LIN {X 0,Y 474.587,Z 340.988,A -85,B 0,C 180,E1 -7401.729,E2 -7401.729} C_VEL
LIN {X 0,Y 474.649,Z 340.986,A -85,B 0,C 180,E1 -7404.494,E2 -7404.494} C_VEL
LIN {X 0,Y 474.672,Z 340.979,A -85,B 0,C 180,E1 -7407.333,E2 -7407.333} C_VEL
LIN {X 0,Y 474.604,Z 340.989,A -85,B 0,C 180,E1 -7410.231,E2 -7410.231} C_VEL
LIN {X 0,Y 474.642,Z 340.983,A -85,B 0,C 180,E1 -7413.221,E2 -7413.221} C_VEL
LIN {X 0,Y 474.592,Z 340.992,A -85,B 0,C 180,E1 -7416.324,E2 -7416.324} C_VEL
LIN {X 0,Y 474.612,Z 340.985,A -85,B 0,C 180,E1 -7419.646,E2 -7419.646} C_VEL
LIN {X 0,Y 474.599,Z 340.99,A -85,B 0,C 180,E1 -7422.234,E2 -7422.234} C_VEL
LIN {X 0,Y 474.616,Z 340.986,A -85,B 0,C 180,E1 -7425.298,E2 -7425.298} C_VEL
LIN {X 0,Y 474.615,Z 340.989,A -85,B 0,C 180,E1 -7428.215,E2 -7428.215} C_VEL
LIN {X 0,Y 474.611,Z 340.986,A -85,B 0,C 180,E1 -7431.543,E2 -7431.543} C_VEL
LIN {X 0,Y 474.623,Z 340.989,A -85,B 0,C 180,E1 -7434.726,E2 -7434.726} C_VEL
LIN {X 0,Y 474.637,Z 340.983,A -85,B 0,C 180,E1 -7437.788,E2 -7437.788} C_VEL
LIN {X 0,Y 474.608,Z 340.989,A -85,B 0,C 180,E1 -7440.889,E2 -7440.889} C_VEL
LIN {X 0,Y 474.612,Z 340.986,A -85,B 0,C 180,E1 -7443.626,E2 -7443.626} C_VEL
LIN {X 0,Y 474.637,Z 340.988,A -85,B 0,C 180,E1 -7446.643,E2 -7446.643} C_VEL
LIN {X 0,Y 474.654,Z 340.984,A -85,B 0,C 180,E1 -7450.09,E2 -7450.09} C_VEL
LIN {X 0,Y 474.642,Z 340.982,A -85,B 0,C 180,E1 -7451.675,E2 -7451.675} C_VEL
LIN {X 0,Y 473.965,Z 341.075,A -85,B 0,C 180,E1 -7452.383,E2 -7452.383} C_VEL
LIN {X 0,Y 471.115,Z 341.424,A -85,B 0,C 180,E1 -7453.534,E2 -7453.534} C_VEL
LIN {X 0,Y 468.709,Z 341.728,A -85,B 0,C 180,E1 -7454.462,E2 -7454.462} C_VEL
LIN {X 0,Y 467.674,Z 341.851,A -85,B 0,C 180,E1 -7455.179,E2 -7455.179} C_VEL
LIN {X 0,Y 467.588,Z 341.86,A -85,B 0,C 180,E1 -7455.422,E2 -7455.422} C_VEL
LIN {X 0,Y 467.653,Z 341.855,A -85,B 0,C 180,E1 -7458.734,E2 -7458.734} C_VEL
LIN {X 0,Y 467.66,Z 341.851,A -85,B 0,C 180,E1 -7461.357,E2 -7461.357} C_VEL
LIN {X 0,Y 467.705,Z 341.85,A -85,B 0,C 180,E1 -7463.963,E2 -7463.963} C_VEL
LIN {X 0,Y 467.817,Z 341.832,A -85,B 0,C 180,E1 -7467.417,E2 -7467.417} C_VEL
LIN {X 0,Y 467.853,Z 341.832,A -85,B 0,C 180,E1 -7470,E2 -7470} C_VEL
LIN {X 0,Y 467.815,Z 341.836,A -85,B 0,C 180,E1 -7472.584,E2 -7472.584} C_VEL
LIN {X 0,Y 467.706,Z 341.852,A -85,B 0,C 180,E1 -7476.038,E2 -7476.038} C_VEL
LIN {X 0,Y 467.637,Z 341.857,A -85,B 0,C 180,E1 -7478.644,E2 -7478.644} C_VEL
LIN {X 0,Y 467.656,Z 341.857,A -85,B 0,C 180,E1 -7482.356,E2 -7482.356} C_VEL
LIN {X 0,Y 467.613,Z 341.978,A -85,B 0,C 180,E1 -7485.194,E2 -7485.194} C_VEL
LIN {X 0,Y 468.283,Z 345.088,A -85,B 0,C 180,E1 -7485.805,E2 -7485.805} C_VEL
LIN {X 0,Y 476.001,Z 364.043,A -85,B 0,C 180,E1 -7486.537,E2 -7486.537} C_VEL
LIN {X 0,Y 474.194,Z 509.031,A -85,B 0,C 180,E1 -7488.849,E2 -7488.849} C_VEL
LIN {X 0,Y 473.785,Z 524.801,A -85,B 0,C 180,E1 -7489.272,E2 -7489.272} C_VEL
LIN {X 0,Y 473.25,Z 539.852,A -85,B 0,C 180,E1 -7489.859,E2 -7489.859} C_VEL
LIN {X 0,Y 472.524,Z 554.963,A -85,B 0,C 180,E1 -7490.645,E2 -7490.645} C_VEL
LIN {X 0,Y 471.782,Z 568.297,A -85,B 0,C 180,E1 -7491.521,E2 -7491.521} C_VEL
LIN {X 0,Y 470.984,Z 580.882,A -85,B 0,C 180,E1 -7492.531,E2 -7492.531} C_VEL
LIN {X 0,Y 470.089,Z 593.972,A -85,B 0,C 180,E1 -7493.808,E2 -7493.808} C_VEL
LIN {X 0,Y 469.383,Z 604.338,A -85,B 0,C 180,E1 -7495.023,E2 -7495.023} C_VEL
LIN {X 0,Y 468.643,Z 615.056,A -85,B 0,C 180,E1 -7496.518,E2 -7496.518} C_VEL
LIN {X 0,Y 468.075,Z 623.773,A -85,B 0,C 180,E1 -7497.983,E2 -7497.983} C_VEL
LIN {X 0,Y 467.53,Z 632.422,A -85,B 0,C 180,E1 -7499.74,E2 -7499.74} C_VEL
LIN {X 0,Y 467.23,Z 638.758,A -85,B 0,C 180,E1 -7501.339,E2 -7501.339} C_VEL
LIN {X 0,Y 466.974,Z 643.497,A -85,B 0,C 180,E1 -7502.807,E2 -7502.807} C_VEL
LIN {X 0,Y 466.851,Z 646.899,A -85,B 0,C 180,E1 -7504.108,E2 -7504.108} C_VEL
LIN {X 0,Y 466.652,Z 650.524,A -85,B 0,C 180,E1 -7505.97,E2 -7505.97} C_VEL
LIN {X 0,Y 466.583,Z 652.01,A -85,B 0,C 180,E1 -7507.05,E2 -7507.05} C_VEL
LIN {X 0,Y 466.575,Z 653.213,A -85,B 0,C 180,E1 -7508.438,E2 -7508.438} C_VEL
LIN {X 0,Y 466.553,Z 653.709,A -85,B 0,C 180,E1 -7510.372,E2 -7510.372} C_VEL
LIN {X 0,Y 466.566,Z 653.334,A -85,B 0,C 180,E1 -7511.513,E2 -7511.513} C_VEL
LIN {X 0,Y 466.619,Z 652.463,A -85,B 0,C 180,E1 -7512.67,E2 -7512.67} C_VEL
LIN {X 0,Y 466.668,Z 651.066,A -85,B 0,C 180,E1 -7513.849,E2 -7513.849} C_VEL
LIN {X 0,Y 466.855,Z 647.895,A -85,B 0,C 180,E1 -7515.607,E2 -7515.607} C_VEL
LIN {X 0,Y 467.042,Z 643.061,A -85,B 0,C 180,E1 -7517.506,E2 -7517.506} C_VEL
LIN {X 0,Y 467.29,Z 637.214,A -85,B 0,C 180,E1 -7519.243,E2 -7519.243} C_VEL
LIN {X 0,Y 467.708,Z 630.356,A -85,B 0,C 180,E1 -7520.867,E2 -7520.867} C_VEL
LIN {X 0,Y 468.244,Z 622.555,A -85,B 0,C 180,E1 -7522.387,E2 -7522.387} C_VEL
LIN {X 0,Y 468.831,Z 613.461,A -85,B 0,C 180,E1 -7523.868,E2 -7523.868} C_VEL
LIN {X 0,Y 469.603,Z 602.591,A -85,B 0,C 180,E1 -7525.34,E2 -7525.34} C_VEL
LIN {X 0,Y 470.454,Z 590.958,A -85,B 0,C 180,E1 -7526.647,E2 -7526.647} C_VEL
LIN {X 0,Y 471.237,Z 578.375,A -85,B 0,C 180,E1 -7527.824,E2 -7527.824} C_VEL
LIN {X 0,Y 472.024,Z 565.723,A -85,B 0,C 180,E1 -7528.798,E2 -7528.798} C_VEL
LIN {X 0,Y 472.796,Z 551.391,A -85,B 0,C 180,E1 -7529.691,E2 -7529.691} C_VEL
LIN {X 0,Y 473.431,Z 537.673,A -85,B 0,C 180,E1 -7530.362,E2 -7530.362} C_VEL
LIN {X 0,Y 473.882,Z 522.925,A -85,B 0,C 180,E1 -7530.909,E2 -7530.909} C_VEL
LIN {X 0,Y 474.283,Z 507.871,A -85,B 0,C 180,E1 -7531.288,E2 -7531.288} C_VEL
LIN {X 0,Y 476.111,Z 364.185,A -85,B 0,C 180,E1 -7533.601,E2 -7533.601} C_VEL
LIN {X 0,Y 468.631,Z 346.42,A -85,B 0,C 180,E1 -7534.341,E2 -7534.341} C_VEL
LIN {X 0,Y 467.593,Z 341.868,A -85,B 0,C 180,E1 -7535.29,E2 -7535.29} C_VEL
LIN {X 0,Y 467.573,Z 341.864,A -85,B 0,C 180,E1 -7538.854,E2 -7538.854} C_VEL
LIN {X 0,Y 467.621,Z 341.863,A -85,B 0,C 180,E1 -7541.602,E2 -7541.602} C_VEL
LIN {X 0,Y 467.598,Z 341.864,A -85,B 0,C 180,E1 -7545.196,E2 -7545.196} C_VEL
LIN {X 0,Y 467.66,Z 341.859,A -85,B 0,C 180,E1 -7547.854,E2 -7547.854} C_VEL
LIN {X 0,Y 467.66,Z 341.857,A -85,B 0,C 180,E1 -7551.356,E2 -7551.356} C_VEL
LIN {X 0,Y 467.706,Z 341.851,A -85,B 0,C 180,E1 -7553.962,E2 -7553.962} C_VEL
LIN {X 0,Y 467.817,Z 341.837,A -85,B 0,C 180,E1 -7557.417,E2 -7557.417} C_VEL
LIN {X 0,Y 467.881,Z 341.829,A -85,B 0,C 180,E1 -7560,E2 -7560} C_VEL
LIN {X 0,Y 467.853,Z 341.828,A -85,B 0,C 180,E1 -7562.583,E2 -7562.583} C_VEL
LIN {X 0,Y 467.715,Z 341.847,A -85,B 0,C 180,E1 -7566.037,E2 -7566.037} C_VEL
LIN {X 0,Y 467.67,Z 341.852,A -85,B 0,C 180,E1 -7568.643,E2 -7568.643} C_VEL
LIN {X 0,Y 467.659,Z 341.852,A -85,B 0,C 180,E1 -7572.145,E2 -7572.145} C_VEL
LIN {X 0,Y 467.641,Z 341.856,A -85,B 0,C 180,E1 -7575.695,E2 -7575.695} C_VEL
LIN {X 0,Y 467.624,Z 341.861,A -85,B 0,C 180,E1 -7579.307,E2 -7579.307} C_VEL
LIN {X 0,Y 467.536,Z 341.868,A -85,B 0,C 180,E1 -7582.073,E2 -7582.073} C_VEL
LIN {X 0,Y 467.603,Z 341.861,A -85,B 0,C 180,E1 -7584.887,E2 -7584.887} C_VEL
LIN {X 0,Y 467.622,Z 341.859,A -85,B 0,C 180,E1 -7587.769,E2 -7587.769} C_VEL
LIN {X 0,Y 467.57,Z 341.87,A -85,B 0,C 180,E1 -7591.045,E2 -7591.045} C_VEL
LIN {X 0,Y 467.589,Z 341.863,A -85,B 0,C 180,E1 -7594.242,E2 -7594.242} C_VEL
LIN {X 0,Y 467.549,Z 341.872,A -85,B 0,C 180,E1 -7597.186,E2 -7597.186} C_VEL
LIN {X 0,Y 467.579,Z 341.865,A -85,B 0,C 180,E1 -7600.264,E2 -7600.264} C_VEL
LIN {X 0,Y 467.588,Z 341.867,A -85,B 0,C 180,E1 -7602.567,E2 -7602.567} C_VEL
LIN {X 0,Y 467.572,Z 341.87,A -85,B 0,C 180,E1 -7605.053,E2 -7605.053} C_VEL
LIN {X 0,Y 467.59,Z 341.865,A -85,B 0,C 180,E1 -7607.44,E2 -7607.44} C_VEL
LIN {X 0,Y 467.583,Z 341.866,A -85,B 0,C 180,E1 -7610.855,E2 -7610.855} C_VEL
LIN {X 0,Y 467.561,Z 341.87,A -85,B 0,C 180,E1 -7614.261,E2 -7614.261} C_VEL
LIN {X 0,Y 467.583,Z 341.869,A -85,B 0,C 180,E1 -7617.321,E2 -7617.321} C_VEL
LIN {X 0,Y 467.59,Z 341.957,A -85,B 0,C 180,E1 -7618.29,E2 -7618.29} C_VEL
LIN {X 0,Y 470.988,Z 355.341,A -85,B 0,C 180,E1 -7620.5,E2 -7620.5} C_VEL
LIN {X 0,Y 472.508,Z 362.159,A -85,B 0,C 180,E1 -7621.578,E2 -7621.578} C_VEL
LIN {X 0,Y 472.251,Z 370.532,A -85,B 0,C 180,E1 -7622.758,E2 -7622.758} C_VEL
LIN {X 0,Y 471.054,Z 392.478,A -85,B 0,C 180,E1 -7625.776,E2 -7625.776} C_VEL
LIN {X 0,Y 471.112,Z 393.337,A -85,B 0,C 180,E1 -7625.837,E2 -7625.837} C_VEL
LIN {X 0,Y 475.725,Z 419.308,A -85,B 0,C 180,E1 -7626.526,E2 -7626.526} C_VEL
LIN {X 0,Y 473.906,Z 560.263,A -85,B 0,C 180,E1 -7628.78,E2 -7628.78} C_VEL
LIN {X 0,Y 473.379,Z 576.364,A -85,B 0,C 180,E1 -7629.212,E2 -7629.212} C_VEL
LIN {X 0,Y 472.664,Z 591.498,A -85,B 0,C 180,E1 -7629.797,E2 -7629.797} C_VEL
LIN {X 0,Y 471.905,Z 605.905,A -85,B 0,C 180,E1 -7630.535,E2 -7630.535} C_VEL
LIN {X 0,Y 471.102,Z 619.398,A -85,B 0,C 180,E1 -7631.405,E2 -7631.405} C_VEL
LIN {X 0,Y 470.194,Z 633.159,A -85,B 0,C 180,E1 -7632.493,E2 -7632.493} C_VEL
LIN {X 0,Y 469.381,Z 645.67,A -85,B 0,C 180,E1 -7633.695,E2 -7633.695} C_VEL
LIN {X 0,Y 468.624,Z 657.082,A -85,B 0,C 180,E1 -7635.007,E2 -7635.007} C_VEL
LIN {X 0,Y 468.004,Z 668.188,A -85,B 0,C 180,E1 -7636.54,E2 -7636.54} C_VEL
LIN {X 0,Y 467.478,Z 677.417,A -85,B 0,C 180,E1 -7638.07,E2 -7638.07} C_VEL
LIN {X 0,Y 467.199,Z 685.087,A -85,B 0,C 180,E1 -7639.6,E2 -7639.6} C_VEL
LIN {X 0,Y 466.898,Z 692.25,A -85,B 0,C 180,E1 -7641.342,E2 -7641.342} C_VEL
LIN {X 0,Y 466.818,Z 697.893,A -85,B 0,C 180,E1 -7643.082,E2 -7643.082} C_VEL
LIN {X 0,Y 466.711,Z 702.161,A -85,B 0,C 180,E1 -7644.816,E2 -7644.816} C_VEL
LIN {X 0,Y 466.708,Z 705.163,A -85,B 0,C 180,E1 -7646.546,E2 -7646.546} C_VEL
LIN {X 0,Y 466.692,Z 706.959,A -85,B 0,C 180,E1 -7648.274,E2 -7648.274} C_VEL
LIN {X 0,Y 466.596,Z 707.583,A -85,B 0,C 180,E1 -7650,E2 -7650} C_VEL
LIN {X 0,Y 466.691,Z 706.998,A -85,B 0,C 180,E1 -7651.726,E2 -7651.726} C_VEL
LIN {X 0,Y 466.707,Z 705.239,A -85,B 0,C 180,E1 -7653.453,E2 -7653.453} C_VEL
LIN {X 0,Y 466.708,Z 702.281,A -85,B 0,C 180,E1 -7655.183,E2 -7655.183} C_VEL
LIN {X 0,Y 466.729,Z 698.058,A -85,B 0,C 180,E1 -7656.918,E2 -7656.918} C_VEL
LIN {X 0,Y 466.898,Z 692.464,A -85,B 0,C 180,E1 -7658.657,E2 -7658.657} C_VEL
LIN {X 0,Y 467.201,Z 685.346,A -85,B 0,C 180,E1 -7660.399,E2 -7660.399} C_VEL
LIN {X 0,Y 467.515,Z 677.733,A -85,B 0,C 180,E1 -7661.929,E2 -7661.929} C_VEL
LIN {X 0,Y 468.043,Z 668.563,A -85,B 0,C 180,E1 -7663.458,E2 -7663.458} C_VEL
LIN {X 0,Y 468.655,Z 657.51,A -85,B 0,C 180,E1 -7664.991,E2 -7664.991} C_VEL
LIN {X 0,Y 469.442,Z 646.16,A -85,B 0,C 180,E1 -7666.302,E2 -7666.302} C_VEL
LIN {X 0,Y 470.221,Z 633.697,A -85,B 0,C 180,E1 -7667.505,E2 -7667.505} C_VEL
LIN {X 0,Y 471.129,Z 619.955,A -85,B 0,C 180,E1 -7668.593,E2 -7668.593} C_VEL
LIN {X 0,Y 471.948,Z 606.475,A -85,B 0,C 180,E1 -7669.462,E2 -7669.462} C_VEL
LIN {X 0,Y 472.758,Z 592.065,A -85,B 0,C 180,E1 -7670.199,E2 -7670.199} C_VEL
LIN {X 0,Y 473.357,Z 576.997,A -85,B 0,C 180,E1 -7670.785,E2 -7670.785} C_VEL
LIN {X 0,Y 473.904,Z 561.89,A -85,B 0,C 180,E1 -7671.191,E2 -7671.191} C_VEL
LIN {X 0,Y 475.392,Z 446.29,A -85,B 0,C 180,E1 -7673.034,E2 -7673.034} C_VEL
LIN {X 0,Y 475.685,Z 419.152,A -85,B 0,C 180,E1 -7673.468,E2 -7673.468} C_VEL
LIN {X 0,Y 471.151,Z 394.04,A -85,B 0,C 180,E1 -7674.124,E2 -7674.124} C_VEL
LIN {X 0,Y 472.402,Z 371.288,A -85,B 0,C 180,E1 -7677.241,E2 -7677.241} C_VEL
LIN {X 0,Y 472.755,Z 362.946,A -85,B 0,C 180,E1 -7678.405,E2 -7678.405} C_VEL
LIN {X 0,Y 468.809,Z 346.686,A -85,B 0,C 180,E1 -7680.998,E2 -7680.998} C_VEL
LIN {X 0,Y 467.572,Z 341.869,A -85,B 0,C 180,E1 -7681.804,E2 -7681.804} C_VEL
LIN {X 0,Y 467.562,Z 341.87,A -85,B 0,C 180,E1 -7684.832,E2 -7684.832} C_VEL
LIN {X 0,Y 467.563,Z 341.87,A -85,B 0,C 180,E1 -7688.044,E2 -7688.044} C_VEL
LIN {X 0,Y 467.579,Z 341.87,A -85,B 0,C 180,E1 -7691.277,E2 -7691.277} C_VEL
LIN {X 0,Y 467.564,Z 341.865,A -85,B 0,C 180,E1 -7693.822,E2 -7693.822} C_VEL
LIN {X 0,Y 467.568,Z 341.863,A -85,B 0,C 180,E1 -7696.257,E2 -7696.257} C_VEL
LIN {X 0,Y 467.579,Z 341.864,A -85,B 0,C 180,E1 -7698.722,E2 -7698.722} C_VEL
LIN {X 0,Y 467.563,Z 341.864,A -85,B 0,C 180,E1 -7701.956,E2 -7701.956} C_VEL
LIN {X 0,Y 467.566,Z 341.872,A -85,B 0,C 180,E1 -7705.168,E2 -7705.168} C_VEL
LIN {X 0,Y 467.579,Z 341.862,A -85,B 0,C 180,E1 -7708.26,E2 -7708.26} C_VEL
LIN {X 0,Y 467.574,Z 341.869,A -85,B 0,C 180,E1 -7711.251,E2 -7711.251} C_VEL
LIN {X 0,Y 467.607,Z 341.858,A -85,B 0,C 180,E1 -7714.16,E2 -7714.16} C_VEL
LIN {X 0,Y 467.574,Z 341.87,A -85,B 0,C 180,E1 -7716.996,E2 -7716.996} C_VEL
LIN {X 0,Y 467.621,Z 341.857,A -85,B 0,C 180,E1 -7719.777,E2 -7719.777} C_VEL
LIN {X 0,Y 467.606,Z 341.86,A -85,B 0,C 180,E1 -7722.507,E2 -7722.507} C_VEL
LIN {X 0,Y 467.605,Z 341.864,A -85,B 0,C 180,E1 -7725.197,E2 -7725.197} C_VEL
LIN {X 0,Y 467.653,Z 341.852,A -85,B 0,C 180,E1 -7727.855,E2 -7727.855} C_VEL
LIN {X 0,Y 467.679,Z 341.852,A -85,B 0,C 180,E1 -7731.357,E2 -7731.357} C_VEL
LIN {X 0,Y 467.732,Z 341.842,A -85,B 0,C 180,E1 -7733.963,E2 -7733.963} C_VEL
LIN {X 0,Y 467.858,Z 341.829,A -85,B 0,C 180,E1 -7737.417,E2 -7737.417} C_VEL
LIN {X 0,Y 467.881,Z 341.824,A -85,B 0,C 180,E1 -7740,E2 -7740} C_VEL
LIN {X 0,Y 467.857,Z 341.831,A -85,B 0,C 180,E1 -7742.583,E2 -7742.583} C_VEL
LIN {X 0,Y 467.744,Z 341.841,A -85,B 0,C 180,E1 -7746.038,E2 -7746.038} C_VEL
LIN {X 0,Y 467.68,Z 341.855,A -85,B 0,C 180,E1 -7748.643,E2 -7748.643} C_VEL
LIN {X 0,Y 467.654,Z 341.853,A -85,B 0,C 180,E1 -7752.146,E2 -7752.146} C_VEL
LIN {X 0,Y 467.637,Z 341.854,A -85,B 0,C 180,E1 -7755.695,E2 -7755.695} C_VEL
LIN {X 0,Y 467.616,Z 341.866,A -85,B 0,C 180,E1 -7758.765,E2 -7758.765} C_VEL
LIN {X 0,Y 467.579,Z 341.864,A -85,B 0,C 180,E1 -7761.269,E2 -7761.269} C_VEL
LIN {X 0,Y 467.567,Z 341.863,A -85,B 0,C 180,E1 -7763.944,E2 -7763.944} C_VEL
LIN {X 0,Y 467.589,Z 341.868,A -85,B 0,C 180,E1 -7766.802,E2 -7766.802} C_VEL
LIN {X 0,Y 467.552,Z 341.865,A -85,B 0,C 180,E1 -7769.739,E2 -7769.739} C_VEL
LIN {X 0,Y 467.582,Z 341.868,A -85,B 0,C 180,E1 -7772.759,E2 -7772.759} C_VEL
LIN {X 0,Y 467.555,Z 341.865,A -85,B 0,C 180,E1 -7775.89,E2 -7775.89} C_VEL
LIN {X 0,Y 467.557,Z 341.866,A -85,B 0,C 180,E1 -7779.148,E2 -7779.148} C_VEL
LIN {X 0,Y 467.572,Z 341.863,A -85,B 0,C 180,E1 -7781.404,E2 -7781.404} C_VEL
LIN {X 0,Y 467.565,Z 341.866,A -85,B 0,C 180,E1 -7785.053,E2 -7785.053} C_VEL
LIN {X 0,Y 467.574,Z 341.87,A -85,B 0,C 180,E1 -7788.597,E2 -7788.597} C_VEL
LIN {X 0,Y 467.563,Z 341.865,A -85,B 0,C 180,E1 -7791.956,E2 -7791.956} C_VEL
LIN {X 0,Y 467.564,Z 341.864,A -85,B 0,C 180,E1 -7795.168,E2 -7795.168} C_VEL
LIN {X 0,Y 467.584,Z 341.866,A -85,B 0,C 180,E1 -7798.261,E2 -7798.261} C_VEL
LIN {X 0,Y 467.557,Z 341.865,A -85,B 0,C 180,E1 -7801.25,E2 -7801.25} C_VEL
LIN {X 0,Y 467.584,Z 341.865,A -85,B 0,C 180,E1 -7804.159,E2 -7804.159} C_VEL
LIN {X 0,Y 467.578,Z 341.863,A -85,B 0,C 180,E1 -7806.996,E2 -7806.996} C_VEL
LIN {X 0,Y 467.623,Z 341.857,A -85,B 0,C 180,E1 -7809.778,E2 -7809.778} C_VEL
LIN {X 0,Y 467.571,Z 341.869,A -85,B 0,C 180,E1 -7812.506,E2 -7812.506} C_VEL
LIN {X 0,Y 467.588,Z 341.86,A -85,B 0,C 180,E1 -7815.422,E2 -7815.422} C_VEL
LIN {X 0,Y 466.921,Z 341.95,A -85,B 0,C 180,E1 -7816.141,E2 -7816.141} C_VEL
LIN {X 0,Y 464.082,Z 342.299,A -85,B 0,C 180,E1 -7817.31,E2 -7817.31} C_VEL
LIN {X 0,Y 461.684,Z 342.603,A -85,B 0,C 180,E1 -7818.252,E2 -7818.252} C_VEL
LIN {X 0,Y 460.657,Z 342.725,A -85,B 0,C 180,E1 -7818.98,E2 -7818.98} C_VEL
LIN {X 0,Y 460.574,Z 342.734,A -85,B 0,C 180,E1 -7819.226,E2 -7819.226} C_VEL
LIN {X 0,Y 460.667,Z 342.727,A -85,B 0,C 180,E1 -7822.594,E2 -7822.594} C_VEL
LIN {X 0,Y 460.677,Z 342.724,A -85,B 0,C 180,E1 -7824.748,E2 -7824.748} C_VEL
LIN {X 0,Y 460.761,Z 342.711,A -85,B 0,C 180,E1 -7827.378,E2 -7827.378} C_VEL
LIN {X 0,Y 460.823,Z 342.708,A -85,B 0,C 180,E1 -7830,E2 -7830} C_VEL
LIN {X 0,Y 460.759,Z 342.714,A -85,B 0,C 180,E1 -7832.623,E2 -7832.623} C_VEL
LIN {X 0,Y 460.672,Z 342.729,A -85,B 0,C 180,E1 -7836.131,E2 -7836.131} C_VEL
LIN {X 0,Y 460.592,Z 342.733,A -85,B 0,C 180,E1 -7838.777,E2 -7838.777} C_VEL
LIN {X 0,Y 460.602,Z 342.735,A -85,B 0,C 180,E1 -7842.435,E2 -7842.435} C_VEL
LIN {X 0,Y 460.552,Z 342.857,A -85,B 0,C 180,E1 -7844.895,E2 -7844.895} C_VEL
LIN {X 0,Y 461.146,Z 345.416,A -85,B 0,C 180,E1 -7845.412,E2 -7845.412} C_VEL
LIN {X 0,Y 469.499,Z 365.897,A -85,B 0,C 180,E1 -7846.226,E2 -7846.226} C_VEL
LIN {X 0,Y 467.558,Z 509.675,A -85,B 0,C 180,E1 -7848.554,E2 -7848.554} C_VEL
LIN {X 0,Y 467.13,Z 525.283,A -85,B 0,C 180,E1 -7848.981,E2 -7848.981} C_VEL
LIN {X 0,Y 466.554,Z 540.472,A -85,B 0,C 180,E1 -7849.583,E2 -7849.583} C_VEL
LIN {X 0,Y 465.902,Z 554.198,A -85,B 0,C 180,E1 -7850.301,E2 -7850.301} C_VEL
LIN {X 0,Y 465.084,Z 567.53,A -85,B 0,C 180,E1 -7851.173,E2 -7851.173} C_VEL
LIN {X 0,Y 464.192,Z 580.845,A -85,B 0,C 180,E1 -7852.242,E2 -7852.242} C_VEL
LIN {X 0,Y 463.362,Z 593.316,A -85,B 0,C 180,E1 -7853.463,E2 -7853.463} C_VEL
LIN {X 0,Y 462.556,Z 603.963,A -85,B 0,C 180,E1 -7854.71,E2 -7854.71} C_VEL
LIN {X 0,Y 461.765,Z 614.583,A -85,B 0,C 180,E1 -7856.192,E2 -7856.192} C_VEL
LIN {X 0,Y 461.203,Z 622.632,A -85,B 0,C 180,E1 -7857.53,E2 -7857.53} C_VEL
LIN {X 0,Y 460.63,Z 631.16,A -85,B 0,C 180,E1 -7859.225,E2 -7859.225} C_VEL
LIN {X 0,Y 460.254,Z 637.429,A -85,B 0,C 180,E1 -7860.735,E2 -7860.735} C_VEL
LIN {X 0,Y 459.985,Z 642.836,A -85,B 0,C 180,E1 -7862.328,E2 -7862.328} C_VEL
LIN {X 0,Y 459.79,Z 646.935,A -85,B 0,C 180,E1 -7863.87,E2 -7863.87} C_VEL
LIN {X 0,Y 459.619,Z 650.289,A -85,B 0,C 180,E1 -7865.525,E2 -7865.525} C_VEL
LIN {X 0,Y 459.48,Z 652.728,A -85,B 0,C 180,E1 -7867.309,E2 -7867.309} C_VEL
LIN {X 0,Y 459.472,Z 653.857,A -85,B 0,C 180,E1 -7868.839,E2 -7868.839} C_VEL
LIN {X 0,Y 459.463,Z 654.164,A -85,B 0,C 180,E1 -7870.11,E2 -7870.11} C_VEL
LIN {X 0,Y 459.478,Z 653.79,A -85,B 0,C 180,E1 -7871.454,E2 -7871.454} C_VEL
LIN {X 0,Y 459.545,Z 652.825,A -85,B 0,C 180,E1 -7872.77,E2 -7872.77} C_VEL
LIN {X 0,Y 459.695,Z 650.23,A -85,B 0,C 180,E1 -7874.69,E2 -7874.69} C_VEL
LIN {X 0,Y 459.889,Z 646.337,A -85,B 0,C 180,E1 -7876.552,E2 -7876.552} C_VEL
LIN {X 0,Y 460.131,Z 640.885,A -85,B 0,C 180,E1 -7878.454,E2 -7878.454} C_VEL
LIN {X 0,Y 460.476,Z 634.689,A -85,B 0,C 180,E1 -7880.131,E2 -7880.131} C_VEL
LIN {X 0,Y 460.892,Z 628.162,A -85,B 0,C 180,E1 -7881.582,E2 -7881.582} C_VEL
LIN {X 0,Y 461.469,Z 620.506,A -85,B 0,C 180,E1 -7883.017,E2 -7883.017} C_VEL
LIN {X 0,Y 462.129,Z 611.26,A -85,B 0,C 180,E1 -7884.473,E2 -7884.473} C_VEL
LIN {X 0,Y 462.951,Z 600.977,A -85,B 0,C 180,E1 -7885.827,E2 -7885.827} C_VEL
LIN {X 0,Y 463.773,Z 589.761,A -85,B 0,C 180,E1 -7887.067,E2 -7887.067} C_VEL
LIN {X 0,Y 464.547,Z 578.052,A -85,B 0,C 180,E1 -7888.155,E2 -7888.155} C_VEL
LIN {X 0,Y 465.38,Z 565.74,A -85,B 0,C 180,E1 -7889.105,E2 -7889.105} C_VEL
LIN {X 0,Y 466.139,Z 551.782,A -85,B 0,C 180,E1 -7889.984,E2 -7889.984} C_VEL
LIN {X 0,Y 466.842,Z 537.238,A -85,B 0,C 180,E1 -7890.699,E2 -7890.699} C_VEL
LIN {X 0,Y 467.344,Z 521.749,A -85,B 0,C 180,E1 -7891.265,E2 -7891.265} C_VEL
LIN {X 0,Y 467.724,Z 506.873,A -85,B 0,C 180,E1 -7891.627,E2 -7891.627} C_VEL
LIN {X 0,Y 469.739,Z 366.212,A -85,B 0,C 180,E1 -7893.922,E2 -7893.922} C_VEL
LIN {X 0,Y 462.361,Z 349.033,A -85,B 0,C 180,E1 -7894.656,E2 -7894.656} C_VEL
LIN {X 0,Y 461.525,Z 346.887,A -85,B 0,C 180,E1 -7894.762,E2 -7894.762} C_VEL
LIN {X 0,Y 460.541,Z 342.744,A -85,B 0,C 180,E1 -7895.667,E2 -7895.667} C_VEL
LIN {X 0,Y 460.52,Z 342.743,A -85,B 0,C 180,E1 -7898.58,E2 -7898.58} C_VEL
LIN {X 0,Y 460.585,Z 342.736,A -85,B 0,C 180,E1 -7901.31,E2 -7901.31} C_VEL
LIN {X 0,Y 460.57,Z 342.742,A -85,B 0,C 180,E1 -7904.057,E2 -7904.057} C_VEL
LIN {X 0,Y 460.613,Z 342.736,A -85,B 0,C 180,E1 -7907.666,E2 -7907.666} C_VEL
LIN {X 0,Y 460.612,Z 342.734,A -85,B 0,C 180,E1 -7911.223,E2 -7911.223} C_VEL
LIN {X 0,Y 460.672,Z 342.729,A -85,B 0,C 180,E1 -7913.869,E2 -7913.869} C_VEL
LIN {X 0,Y 460.761,Z 342.716,A -85,B 0,C 180,E1 -7917.377,E2 -7917.377} C_VEL
LIN {X 0,Y 460.851,Z 342.704,A -85,B 0,C 180,E1 -7920,E2 -7920} C_VEL
LIN {X 0,Y 460.794,Z 342.708,A -85,B 0,C 180,E1 -7922.622,E2 -7922.622} C_VEL
LIN {X 0,Y 460.68,Z 342.723,A -85,B 0,C 180,E1 -7926.13,E2 -7926.13} C_VEL
LIN {X 0,Y 460.62,Z 342.731,A -85,B 0,C 180,E1 -7928.776,E2 -7928.776} C_VEL
LIN {X 0,Y 460.616,Z 342.729,A -85,B 0,C 180,E1 -7932.445,E2 -7932.445} C_VEL
LIN {X 0,Y 460.603,Z 342.731,A -85,B 0,C 180,E1 -7935.997,E2 -7935.997} C_VEL
LIN {X 0,Y 460.57,Z 342.74,A -85,B 0,C 180,E1 -7939.615,E2 -7939.615} C_VEL
LIN {X 0,Y 460.512,Z 342.743,A -85,B 0,C 180,E1 -7942.428,E2 -7942.428} C_VEL
LIN {X 0,Y 460.57,Z 342.738,A -85,B 0,C 180,E1 -7945.802,E2 -7945.802} C_VEL
LIN {X 0,Y 460.554,Z 342.738,A -85,B 0,C 180,E1 -7948.233,E2 -7948.233} C_VEL
LIN {X 0,Y 460.523,Z 342.747,A -85,B 0,C 180,E1 -7951.283,E2 -7951.283} C_VEL
LIN {X 0,Y 460.533,Z 342.743,A -85,B 0,C 180,E1 -7954.505,E2 -7954.505} C_VEL
LIN {X 0,Y 460.502,Z 342.748,A -85,B 0,C 180,E1 -7957.623,E2 -7957.623} C_VEL
LIN {X 0,Y 460.543,Z 342.742,A -85,B 0,C 180,E1 -7960.269,E2 -7960.269} C_VEL
LIN {X 0,Y 460.502,Z 342.749,A -85,B 0,C 180,E1 -7963.375,E2 -7963.375} C_VEL
LIN {X 0,Y 460.51,Z 342.748,A -85,B 0,C 180,E1 -7966.625,E2 -7966.625} C_VEL
LIN {X 0,Y 460.544,Z 342.743,A -85,B 0,C 180,E1 -7969.73,E2 -7969.73} C_VEL
LIN {X 0,Y 460.527,Z 342.749,A -85,B 0,C 180,E1 -7972.519,E2 -7972.519} C_VEL
LIN {X 0,Y 460.547,Z 342.743,A -85,B 0,C 180,E1 -7975.623,E2 -7975.623} C_VEL
LIN {X 0,Y 460.573,Z 342.841,A -85,B 0,C 180,E1 -7977.927,E2 -7977.927} C_VEL
LIN {X 0,Y 464.108,Z 356.713,A -85,B 0,C 180,E1 -7980.268,E2 -7980.268} C_VEL
LIN {X 0,Y 465.66,Z 363.48,A -85,B 0,C 180,E1 -7981.363,E2 -7981.363} C_VEL
LIN {X 0,Y 465.683,Z 368.551,A -85,B 0,C 180,E1 -7982.105,E2 -7982.105} C_VEL
LIN {X 0,Y 464.362,Z 390.424,A -85,B 0,C 180,E1 -7985.166,E2 -7985.166} C_VEL
LIN {X 0,Y 464.282,Z 392.309,A -85,B 0,C 180,E1 -7985.429,E2 -7985.429} C_VEL
LIN {X 0,Y 469.206,Z 420.118,A -85,B 0,C 180,E1 -7986.191,E2 -7986.191} C_VEL
LIN {X 0,Y 467.501,Z 547.155,A -85,B 0,C 180,E1 -7988.243,E2 -7988.243} C_VEL
LIN {X 0,Y 467.162,Z 564.361,A -85,B 0,C 180,E1 -7988.574,E2 -7988.574} C_VEL
LIN {X 0,Y 466.567,Z 579.856,A -85,B 0,C 180,E1 -7989.044,E2 -7989.044} C_VEL
LIN {X 0,Y 465.835,Z 593.897,A -85,B 0,C 180,E1 -7989.634,E2 -7989.634} C_VEL
LIN {X 0,Y 464.933,Z 609.002,A -85,B 0,C 180,E1 -7990.461,E2 -7990.461} C_VEL
LIN {X 0,Y 463.969,Z 623.292,A -85,B 0,C 180,E1 -7991.452,E2 -7991.452} C_VEL
LIN {X 0,Y 463.078,Z 636.278,A -85,B 0,C 180,E1 -7992.558,E2 -7992.558} C_VEL
LIN {X 0,Y 462.358,Z 647.201,A -85,B 0,C 180,E1 -7993.667,E2 -7993.667} C_VEL
LIN {X 0,Y 461.54,Z 658.296,A -85,B 0,C 180,E1 -7994.997,E2 -7994.997} C_VEL
LIN {X 0,Y 460.929,Z 669.114,A -85,B 0,C 180,E1 -7996.554,E2 -7996.554} C_VEL
LIN {X 0,Y 460.406,Z 678.194,A -85,B 0,C 180,E1 -7998.121,E2 -7998.121} C_VEL
LIN {X 0,Y 460.127,Z 684.64,A -85,B 0,C 180,E1 -7999.438,E2 -7999.438} C_VEL
LIN {X 0,Y 459.834,Z 691.812,A -85,B 0,C 180,E1 -8001.208,E2 -8001.208} C_VEL
LIN {X 0,Y 459.727,Z 697.463,A -85,B 0,C 180,E1 -8002.975,E2 -8002.975} C_VEL
LIN {X 0,Y 459.619,Z 701.738,A -85,B 0,C 180,E1 -8004.736,E2 -8004.736} C_VEL
LIN {X 0,Y 459.62,Z 704.746,A -85,B 0,C 180,E1 -8006.493,E2 -8006.493} C_VEL
LIN {X 0,Y 459.629,Z 706.549,A -85,B 0,C 180,E1 -8008.247,E2 -8008.247} C_VEL
LIN {X 0,Y 459.527,Z 707.175,A -85,B 0,C 180,E1 -8010,E2 -8010} C_VEL
LIN {X 0,Y 459.628,Z 706.592,A -85,B 0,C 180,E1 -8011.752,E2 -8011.752} C_VEL
LIN {X 0,Y 459.619,Z 704.83,A -85,B 0,C 180,E1 -8013.506,E2 -8013.506} C_VEL
LIN {X 0,Y 459.615,Z 701.87,A -85,B 0,C 180,E1 -8015.264,E2 -8015.264} C_VEL
LIN {X 0,Y 459.652,Z 697.643,A -85,B 0,C 180,E1 -8017.026,E2 -8017.026} C_VEL
LIN {X 0,Y 459.833,Z 692.043,A -85,B 0,C 180,E1 -8018.791,E2 -8018.791} C_VEL
LIN {X 0,Y 460.13,Z 684.917,A -85,B 0,C 180,E1 -8020.561,E2 -8020.561} C_VEL
LIN {X 0,Y 460.482,Z 677.294,A -85,B 0,C 180,E1 -8022.113,E2 -8022.113} C_VEL
LIN {X 0,Y 461.051,Z 668.111,A -85,B 0,C 180,E1 -8023.666,E2 -8023.666} C_VEL
LIN {X 0,Y 461.712,Z 657.035,A -85,B 0,C 180,E1 -8025.222,E2 -8025.222} C_VEL
LIN {X 0,Y 462.539,Z 645.665,A -85,B 0,C 180,E1 -8026.552,E2 -8026.552} C_VEL
LIN {X 0,Y 463.308,Z 633.177,A -85,B 0,C 180,E1 -8027.775,E2 -8027.775} C_VEL
LIN {X 0,Y 464.359,Z 619.409,A -85,B 0,C 180,E1 -8028.875,E2 -8028.875} C_VEL
LIN {X 0,Y 465.189,Z 605.901,A -85,B 0,C 180,E1 -8029.757,E2 -8029.757} C_VEL
LIN {X 0,Y 466.03,Z 591.884,A -85,B 0,C 180,E1 -8030.482,E2 -8030.482} C_VEL
LIN {X 0,Y 466.714,Z 576.352,A -85,B 0,C 180,E1 -8031.093,E2 -8031.093} C_VEL
LIN {X 0,Y 467.254,Z 561.022,A -85,B 0,C 180,E1 -8031.507,E2 -8031.507} C_VEL
LIN {X 0,Y 469.028,Z 431.404,A -85,B 0,C 180,E1 -8033.601,E2 -8033.601} C_VEL
LIN {X 0,Y 469.031,Z 419.626,A -85,B 0,C 180,E1 -8033.8,E2 -8033.8} C_VEL
LIN {X 0,Y 464.389,Z 393.575,A -85,B 0,C 180,E1 -8034.504,E2 -8034.504} C_VEL
LIN {X 0,Y 465.595,Z 372.672,A -85,B 0,C 180,E1 -8037.411,E2 -8037.411} C_VEL
LIN {X 0,Y 465.989,Z 364.902,A -85,B 0,C 180,E1 -8038.51,E2 -8038.51} C_VEL
LIN {X 0,Y 461.89,Z 347.962,A -85,B 0,C 180,E1 -8041.254,E2 -8041.254} C_VEL
LIN {X 0,Y 460.544,Z 342.742,A -85,B 0,C 180,E1 -8042.166,E2 -8042.166} C_VEL
LIN {X 0,Y 460.508,Z 342.748,A -85,B 0,C 180,E1 -8045.445,E2 -8045.445} C_VEL
LIN {X 0,Y 460.542,Z 342.748,A -85,B 0,C 180,E1 -8048.898,E2 -8048.898} C_VEL
LIN {X 0,Y 460.521,Z 342.741,A -85,B 0,C 180,E1 -8052.181,E2 -8052.181} C_VEL
LIN {X 0,Y 460.518,Z 342.747,A -85,B 0,C 180,E1 -8055.412,E2 -8055.412} C_VEL
LIN {X 0,Y 460.532,Z 342.74,A -85,B 0,C 180,E1 -8058.397,E2 -8058.397} C_VEL
LIN {X 0,Y 460.523,Z 342.748,A -85,B 0,C 180,E1 -8061.267,E2 -8061.267} C_VEL
LIN {X 0,Y 460.511,Z 342.743,A -85,B 0,C 180,E1 -8064.555,E2 -8064.555} C_VEL
LIN {X 0,Y 460.528,Z 342.741,A -85,B 0,C 180,E1 -8067.716,E2 -8067.716} C_VEL
LIN {X 0,Y 460.537,Z 342.742,A -85,B 0,C 180,E1 -8070.769,E2 -8070.769} C_VEL
LIN {X 0,Y 460.56,Z 342.737,A -85,B 0,C 180,E1 -8073.735,E2 -8073.735} C_VEL
LIN {X 0,Y 460.543,Z 342.741,A -85,B 0,C 180,E1 -8076.624,E2 -8076.624} C_VEL
LIN {X 0,Y 460.549,Z 342.74,A -85,B 0,C 180,E1 -8079.453,E2 -8079.453} C_VEL
LIN {X 0,Y 460.556,Z 342.737,A -85,B 0,C 180,E1 -8082.23,E2 -8082.23} C_VEL
LIN {X 0,Y 460.563,Z 342.743,A -85,B 0,C 180,E1 -8084.965,E2 -8084.965} C_VEL
LIN {X 0,Y 460.608,Z 342.733,A -85,B 0,C 180,E1 -8088.56,E2 -8088.56} C_VEL
LIN {X 0,Y 460.692,Z 342.72,A -85,B 0,C 180,E1 -8092.109,E2 -8092.109} C_VEL
LIN {X 0,Y 460.692,Z 342.725,A -85,B 0,C 180,E1 -8094.749,E2 -8094.749} C_VEL
LIN {X 0,Y 460.823,Z 342.706,A -85,B 0,C 180,E1 -8097.378,E2 -8097.378} C_VEL
LIN {X 0,Y 460.851,Z 342.7,A -85,B 0,C 180,E1 -8100,E2 -8100} C_VEL
LIN {X 0,Y 460.822,Z 342.708,A -85,B 0,C 180,E1 -8102.623,E2 -8102.623} C_VEL
LIN {X 0,Y 460.71,Z 342.718,A -85,B 0,C 180,E1 -8106.13,E2 -8106.13} C_VEL
LIN {X 0,Y 460.627,Z 342.735,A -85,B 0,C 180,E1 -8108.777,E2 -8108.777} C_VEL
LIN {X 0,Y 460.611,Z 342.733,A -85,B 0,C 180,E1 -8112.445,E2 -8112.445} C_VEL
LIN {X 0,Y 460.598,Z 342.731,A -85,B 0,C 180,E1 -8115.998,E2 -8115.998} C_VEL
LIN {X 0,Y 460.569,Z 342.741,A -85,B 0,C 180,E1 -8118.902,E2 -8118.902} C_VEL
LIN {X 0,Y 460.514,Z 342.742,A -85,B 0,C 180,E1 -8121.486,E2 -8121.486} C_VEL
LIN {X 0,Y 460.534,Z 342.742,A -85,B 0,C 180,E1 -8124.333,E2 -8124.333} C_VEL
LIN {X 0,Y 460.576,Z 342.734,A -85,B 0,C 180,E1 -8127.746,E2 -8127.746} C_VEL
LIN {X 0,Y 460.536,Z 342.74,A -85,B 0,C 180,E1 -8131.256,E2 -8131.256} C_VEL
LIN {X 0,Y 460.533,Z 342.745,A -85,B 0,C 180,E1 -8134.506,E2 -8134.506} C_VEL
LIN {X 0,Y 460.501,Z 342.743,A -85,B 0,C 180,E1 -8137.624,E2 -8137.624} C_VEL
LIN {X 0,Y 460.536,Z 342.743,A -85,B 0,C 180,E1 -8140.269,E2 -8140.269} C_VEL
LIN {X 0,Y 460.508,Z 342.743,A -85,B 0,C 180,E1 -8143.375,E2 -8143.375} C_VEL
LIN {X 0,Y 460.509,Z 342.75,A -85,B 0,C 180,E1 -8146.626,E2 -8146.626} C_VEL
LIN {X 0,Y 460.535,Z 342.739,A -85,B 0,C 180,E1 -8149.732,E2 -8149.732} C_VEL
LIN {X 0,Y 460.498,Z 342.752,A -85,B 0,C 180,E1 -8152.525,E2 -8152.525} C_VEL
LIN {X 0,Y 460.547,Z 342.738,A -85,B 0,C 180,E1 -8155.624,E2 -8155.624} C_VEL
LIN {X 0,Y 460.539,Z 342.743,A -85,B 0,C 180,E1 -8158.745,E2 -8158.745} C_VEL
LIN {X 0,Y 460.553,Z 342.742,A -85,B 0,C 180,E1 -8162.262,E2 -8162.262} C_VEL
LIN {X 0,Y 460.536,Z 342.744,A -85,B 0,C 180,E1 -8164.705,E2 -8164.705} C_VEL
LIN {X 0,Y 460.513,Z 342.742,A -85,B 0,C 180,E1 -8167.572,E2 -8167.572} C_VEL
LIN {X 0,Y 460.569,Z 342.743,A -85,B 0,C 180,E1 -8170.385,E2 -8170.385} C_VEL
LIN {X 0,Y 460.569,Z 342.739,A -85,B 0,C 180,E1 -8174.058,E2 -8174.058} C_VEL
LIN {X 0,Y 460.613,Z 342.73,A -85,B 0,C 180,E1 -8177.666,E2 -8177.666} C_VEL
LIN {X 0,Y 460.574,Z 342.734,A -85,B 0,C 180,E1 -8179.226,E2 -8179.226} C_VEL
LIN {X 0,Y 459.911,Z 342.822,A -85,B 0,C 180,E1 -8179.956,E2 -8179.956} C_VEL
LIN {X 0,Y 457.071,Z 343.173,A -85,B 0,C 180,E1 -8181.142,E2 -8181.142} C_VEL
LIN {X 0,Y 454.678,Z 343.474,A -85,B 0,C 180,E1 -8182.098,E2 -8182.098} C_VEL
LIN {X 0,Y 453.665,Z 343.597,A -85,B 0,C 180,E1 -8182.837,E2 -8182.837} C_VEL
LIN {X 0,Y 453.589,Z 343.605,A -85,B 0,C 180,E1 -8183.087,E2 -8183.087} C_VEL
LIN {X 0,Y 453.65,Z 343.6,A -85,B 0,C 180,E1 -8184.667,E2 -8184.667} C_VEL
LIN {X 0,Y 453.692,Z 343.599,A -85,B 0,C 180,E1 -8188.225,E2 -8188.225} C_VEL
LIN {X 0,Y 453.771,Z 343.586,A -85,B 0,C 180,E1 -8190,E2 -8190} C_VEL
LIN {X 0,Y 453.706,Z 343.593,A -85,B 0,C 180,E1 -8192.664,E2 -8192.664} C_VEL
LIN {X 0,Y 453.64,Z 343.606,A -85,B 0,C 180,E1 -8196.226,E2 -8196.226} C_VEL
LIN {X 0,Y 453.562,Z 343.608,A -85,B 0,C 180,E1 -8198.914,E2 -8198.914} C_VEL
LIN {X 0,Y 453.569,Z 343.61,A -85,B 0,C 180,E1 -8202.529,E2 -8202.529} C_VEL
LIN {X 0,Y 453.51,Z 343.746,A -85,B 0,C 180,E1 -8204.586,E2 -8204.586} C_VEL
LIN {X 0,Y 453.968,Z 345.775,A -85,B 0,C 180,E1 -8205.001,E2 -8205.001} C_VEL
LIN {X 0,Y 462.998,Z 367.574,A -85,B 0,C 180,E1 -8205.903,E2 -8205.903} C_VEL
LIN {X 0,Y 460.899,Z 510.698,A -85,B 0,C 180,E1 -8208.259,E2 -8208.259} C_VEL
LIN {X 0,Y 460.487,Z 526.088,A -85,B 0,C 180,E1 -8208.694,E2 -8208.694} C_VEL
LIN {X 0,Y 459.931,Z 540.242,A -85,B 0,C 180,E1 -8209.261,E2 -8209.261} C_VEL
LIN {X 0,Y 459.177,Z 554.775,A -85,B 0,C 180,E1 -8210.027,E2 -8210.027} C_VEL
LIN {X 0,Y 458.243,Z 569.439,A -85,B 0,C 180,E1 -8211.012,E2 -8211.012} C_VEL
LIN {X 0,Y 457.321,Z 582.701,A -85,B 0,C 180,E1 -8212.118,E2 -8212.118} C_VEL
LIN {X 0,Y 456.433,Z 594.751,A -85,B 0,C 180,E1 -8213.335,E2 -8213.335} C_VEL
LIN {X 0,Y 455.594,Z 605.361,A -85,B 0,C 180,E1 -8214.614,E2 -8214.614} C_VEL
LIN {X 0,Y 454.865,Z 614.79,A -85,B 0,C 180,E1 -8215.962,E2 -8215.962} C_VEL
LIN {X 0,Y 454.235,Z 623.347,A -85,B 0,C 180,E1 -8217.407,E2 -8217.407} C_VEL
LIN {X 0,Y 453.663,Z 631.06,A -85,B 0,C 180,E1 -8218.955,E2 -8218.955} C_VEL
LIN {X 0,Y 453.211,Z 638.473,A -85,B 0,C 180,E1 -8220.78,E2 -8220.78} C_VEL
LIN {X 0,Y 452.926,Z 643.666,A -85,B 0,C 180,E1 -8222.367,E2 -8222.367} C_VEL
LIN {X 0,Y 452.7,Z 647.808,A -85,B 0,C 180,E1 -8223.979,E2 -8223.979} C_VEL
LIN {X 0,Y 452.594,Z 650.039,A -85,B 0,C 180,E1 -8225.068,E2 -8225.068} C_VEL
LIN {X 0,Y 452.48,Z 651.819,A -85,B 0,C 180,E1 -8226.173,E2 -8226.173} C_VEL
LIN {X 0,Y 452.405,Z 653.43,A -85,B 0,C 180,E1 -8227.601,E2 -8227.601} C_VEL
LIN {X 0,Y 452.382,Z 654.489,A -85,B 0,C 180,E1 -8229.566,E2 -8229.566} C_VEL
LIN {X 0,Y 452.368,Z 654.476,A -85,B 0,C 180,E1 -8230.732,E2 -8230.732} C_VEL
LIN {X 0,Y 452.409,Z 653.98,A -85,B 0,C 180,E1 -8231.912,E2 -8231.912} C_VEL
LIN {X 0,Y 452.479,Z 652.95,A -85,B 0,C 180,E1 -8233.112,E2 -8233.112} C_VEL
LIN {X 0,Y 452.653,Z 650.34,A -85,B 0,C 180,E1 -8234.955,E2 -8234.955} C_VEL
LIN {X 0,Y 452.872,Z 646.091,A -85,B 0,C 180,E1 -8236.935,E2 -8236.935} C_VEL
LIN {X 0,Y 453.121,Z 640.761,A -85,B 0,C 180,E1 -8238.762,E2 -8238.762} C_VEL
LIN {X 0,Y 453.554,Z 634.057,A -85,B 0,C 180,E1 -8240.556,E2 -8240.556} C_VEL
LIN {X 0,Y 454.175,Z 625.846,A -85,B 0,C 180,E1 -8242.319,E2 -8242.319} C_VEL
LIN {X 0,Y 454.921,Z 615.914,A -85,B 0,C 180,E1 -8244.051,E2 -8244.051} C_VEL
LIN {X 0,Y 455.711,Z 606.086,A -85,B 0,C 180,E1 -8245.475,E2 -8245.475} C_VEL
LIN {X 0,Y 456.673,Z 594.377,A -85,B 0,C 180,E1 -8246.884,E2 -8246.884} C_VEL
LIN {X 0,Y 457.558,Z 581.833,A -85,B 0,C 180,E1 -8248.137,E2 -8248.137} C_VEL
LIN {X 0,Y 458.44,Z 569.613,A -85,B 0,C 180,E1 -8249.148,E2 -8249.148} C_VEL
LIN {X 0,Y 459.396,Z 555.058,A -85,B 0,C 180,E1 -8250.121,E2 -8250.121} C_VEL
LIN {X 0,Y 460.035,Z 541.209,A -85,B 0,C 180,E1 -8250.859,E2 -8250.859} C_VEL
LIN {X 0,Y 460.673,Z 525.564,A -85,B 0,C 180,E1 -8251.48,E2 -8251.48} C_VEL
LIN {X 0,Y 461.113,Z 510.898,A -85,B 0,C 180,E1 -8251.884,E2 -8251.884} C_VEL
LIN {X 0,Y 463.286,Z 368.032,A -85,B 0,C 180,E1 -8254.263,E2 -8254.263} C_VEL
LIN {X 0,Y 455.571,Z 350.097,A -85,B 0,C 180,E1 -8255.056,E2 -8255.056} C_VEL
LIN {X 0,Y 454.406,Z 347.349,A -85,B 0,C 180,E1 -8255.207,E2 -8255.207} C_VEL
LIN {X 0,Y 453.514,Z 343.62,A -85,B 0,C 180,E1 -8256.028,E2 -8256.028} C_VEL
LIN {X 0,Y 453.474,Z 343.621,A -85,B 0,C 180,E1 -8259.117,E2 -8259.117} C_VEL
LIN {X 0,Y 453.49,Z 343.623,A -85,B 0,C 180,E1 -8261.943,E2 -8261.943} C_VEL
LIN {X 0,Y 453.523,Z 343.616,A -85,B 0,C 180,E1 -8264.725,E2 -8264.725} C_VEL
LIN {X 0,Y 453.561,Z 343.612,A -85,B 0,C 180,E1 -8268.379,E2 -8268.379} C_VEL
LIN {X 0,Y 453.58,Z 343.609,A -85,B 0,C 180,E1 -8271.086,E2 -8271.086} C_VEL
LIN {X 0,Y 453.639,Z 343.606,A -85,B 0,C 180,E1 -8273.774,E2 -8273.774} C_VEL
LIN {X 0,Y 453.708,Z 343.594,A -85,B 0,C 180,E1 -8277.336,E2 -8277.336} C_VEL
LIN {X 0,Y 453.82,Z 343.58,A -85,B 0,C 180,E1 -8280,E2 -8280} C_VEL
LIN {X 0,Y 453.738,Z 343.587,A -85,B 0,C 180,E1 -8282.663,E2 -8282.663} C_VEL
LIN {X 0,Y 453.646,Z 343.599,A -85,B 0,C 180,E1 -8286.225,E2 -8286.225} C_VEL
LIN {X 0,Y 453.586,Z 343.609,A -85,B 0,C 180,E1 -8288.913,E2 -8288.913} C_VEL
LIN {X 0,Y 453.566,Z 343.608,A -85,B 0,C 180,E1 -8292.528,E2 -8292.528} C_VEL
LIN {X 0,Y 453.547,Z 343.609,A -85,B 0,C 180,E1 -8296.196,E2 -8296.196} C_VEL
LIN {X 0,Y 453.52,Z 343.615,A -85,B 0,C 180,E1 -8299.039,E2 -8299.039} C_VEL
LIN {X 0,Y 453.478,Z 343.62,A -85,B 0,C 180,E1 -8301.836,E2 -8301.836} C_VEL
LIN {X 0,Y 453.514,Z 343.615,A -85,B 0,C 180,E1 -8304.734,E2 -8304.734} C_VEL
LIN {X 0,Y 453.534,Z 343.613,A -85,B 0,C 180,E1 -8307.959,E2 -8307.959} C_VEL
LIN {X 0,Y 453.467,Z 343.623,A -85,B 0,C 180,E1 -8311.525,E2 -8311.525} C_VEL
LIN {X 0,Y 453.489,Z 343.622,A -85,B 0,C 180,E1 -8314.777,E2 -8314.777} C_VEL
LIN {X 0,Y 453.466,Z 343.624,A -85,B 0,C 180,E1 -8318.311,E2 -8318.311} C_VEL
LIN {X 0,Y 453.495,Z 343.623,A -85,B 0,C 180,E1 -8320.609,E2 -8320.609} C_VEL
LIN {X 0,Y 453.458,Z 343.627,A -85,B 0,C 180,E1 -8323.244,E2 -8323.244} C_VEL
LIN {X 0,Y 453.475,Z 343.622,A -85,B 0,C 180,E1 -8325.78,E2 -8325.78} C_VEL
LIN {X 0,Y 453.483,Z 343.622,A -85,B 0,C 180,E1 -8328.209,E2 -8328.209} C_VEL
LIN {X 0,Y 453.517,Z 343.618,A -85,B 0,C 180,E1 -8330.79,E2 -8330.79} C_VEL
LIN {X 0,Y 453.455,Z 343.625,A -85,B 0,C 180,E1 -8333.917,E2 -8333.917} C_VEL
LIN {X 0,Y 453.485,Z 343.625,A -85,B 0,C 180,E1 -8337.151,E2 -8337.151} C_VEL
LIN {X 0,Y 453.525,Z 343.734,A -85,B 0,C 180,E1 -8337.55,E2 -8337.55} C_VEL
LIN {X 0,Y 457.226,Z 358.208,A -85,B 0,C 180,E1 -8340.048,E2 -8340.048} C_VEL
LIN {X 0,Y 459.057,Z 366.987,A -85,B 0,C 180,E1 -8341.478,E2 -8341.478} C_VEL
LIN {X 0,Y 457.834,Z 386.684,A -85,B 0,C 180,E1 -8344.3,E2 -8344.3} C_VEL
LIN {X 0,Y 457.527,Z 392.017,A -85,B 0,C 180,E1 -8345.036,E2 -8345.036} C_VEL
LIN {X 0,Y 462.771,Z 421.63,A -85,B 0,C 180,E1 -8345.864,E2 -8345.864} C_VEL
LIN {X 0,Y 460.708,Z 559.329,A -85,B 0,C 180,E1 -8348.141,E2 -8348.141} C_VEL
LIN {X 0,Y 460.066,Z 575.507,A -85,B 0,C 180,E1 -8348.585,E2 -8348.585} C_VEL
LIN {X 0,Y 459.327,Z 590.229,A -85,B 0,C 180,E1 -8349.168,E2 -8349.168} C_VEL
LIN {X 0,Y 458.445,Z 604.966,A -85,B 0,C 180,E1 -8349.939,E2 -8349.939} C_VEL
LIN {X 0,Y 457.505,Z 618.467,A -85,B 0,C 180,E1 -8350.831,E2 -8350.831} C_VEL
LIN {X 0,Y 456.497,Z 632.238,A -85,B 0,C 180,E1 -8351.95,E2 -8351.95} C_VEL
LIN {X 0,Y 455.617,Z 644.251,A -85,B 0,C 180,E1 -8353.134,E2 -8353.134} C_VEL
LIN {X 0,Y 454.737,Z 656.17,A -85,B 0,C 180,E1 -8354.538,E2 -8354.538} C_VEL
LIN {X 0,Y 453.988,Z 667.283,A -85,B 0,C 180,E1 -8356.116,E2 -8356.116} C_VEL
LIN {X 0,Y 453.336,Z 676.777,A -85,B 0,C 180,E1 -8357.741,E2 -8357.741} C_VEL
LIN {X 0,Y 453.083,Z 684.2,A -85,B 0,C 180,E1 -8359.272,E2 -8359.272} C_VEL
LIN {X 0,Y 452.74,Z 691.378,A -85,B 0,C 180,E1 -8361.069,E2 -8361.069} C_VEL
LIN {X 0,Y 452.646,Z 697.037,A -85,B 0,C 180,E1 -8362.864,E2 -8362.864} C_VEL
LIN {X 0,Y 452.531,Z 701.318,A -85,B 0,C 180,E1 -8364.653,E2 -8364.653} C_VEL
LIN {X 0,Y 452.518,Z 704.33,A -85,B 0,C 180,E1 -8366.438,E2 -8366.438} C_VEL
LIN {X 0,Y 452.538,Z 706.137,A -85,B 0,C 180,E1 -8368.22,E2 -8368.22} C_VEL
LIN {X 0,Y 452.461,Z 706.767,A -85,B 0,C 180,E1 -8370,E2 -8370} C_VEL
LIN {X 0,Y 452.536,Z 706.184,A -85,B 0,C 180,E1 -8371.78,E2 -8371.78} C_VEL
LIN {X 0,Y 452.517,Z 704.42,A -85,B 0,C 180,E1 -8373.561,E2 -8373.561} C_VEL
LIN {X 0,Y 452.528,Z 701.457,A -85,B 0,C 180,E1 -8375.346,E2 -8375.346} C_VEL
LIN {X 0,Y 452.574,Z 697.224,A -85,B 0,C 180,E1 -8377.136,E2 -8377.136} C_VEL
LIN {X 0,Y 452.74,Z 691.614,A -85,B 0,C 180,E1 -8378.93,E2 -8378.93} C_VEL
LIN {X 0,Y 453.088,Z 684.477,A -85,B 0,C 180,E1 -8380.727,E2 -8380.727} C_VEL
LIN {X 0,Y 453.481,Z 675.862,A -85,B 0,C 180,E1 -8382.482,E2 -8382.482} C_VEL
LIN {X 0,Y 454.142,Z 666.153,A -85,B 0,C 180,E1 -8384.107,E2 -8384.107} C_VEL
LIN {X 0,Y 454.767,Z 656.555,A -85,B 0,C 180,E1 -8385.461,E2 -8385.461} C_VEL
LIN {X 0,Y 455.596,Z 645.892,A -85,B 0,C 180,E1 -8386.729,E2 -8386.729} C_VEL
LIN {X 0,Y 456.511,Z 632.639,A -85,B 0,C 180,E1 -8388.048,E2 -8388.048} C_VEL
LIN {X 0,Y 457.443,Z 620.331,A -85,B 0,C 180,E1 -8389.055,E2 -8389.055} C_VEL
LIN {X 0,Y 458.326,Z 607.068,A -85,B 0,C 180,E1 -8389.948,E2 -8389.948} C_VEL
LIN {X 0,Y 459.249,Z 592.766,A -85,B 0,C 180,E1 -8390.716,E2 -8390.716} C_VEL
LIN {X 0,Y 459.912,Z 578.209,A -85,B 0,C 180,E1 -8391.318,E2 -8391.318} C_VEL
LIN {X 0,Y 460.535,Z 563.443,A -85,B 0,C 180,E1 -8391.749,E2 -8391.749} C_VEL
LIN {X 0,Y 460.953,Z 541.908,A -85,B 0,C 180,E1 -8392.14,E2 -8392.14} C_VEL
LIN {X 0,Y 462.501,Z 429.542,A -85,B 0,C 180,E1 -8393.969,E2 -8393.969} C_VEL
LIN {X 0,Y 462.43,Z 420.126,A -85,B 0,C 180,E1 -8394.135,E2 -8394.135} C_VEL
LIN {X 0,Y 457.631,Z 393.22,A -85,B 0,C 180,E1 -8394.877,E2 -8394.877} C_VEL
LIN {X 0,Y 459.028,Z 370.547,A -85,B 0,C 180,E1 -8398.086,E2 -8398.086} C_VEL
LIN {X 0,Y 459.042,Z 366.137,A -85,B 0,C 180,E1 -8398.732,E2 -8398.732} C_VEL
LIN {X 0,Y 455.253,Z 350.405,A -85,B 0,C 180,E1 -8401.321,E2 -8401.321} C_VEL
LIN {X 0,Y 453.497,Z 343.62,A -85,B 0,C 180,E1 -8402.517,E2 -8402.517} C_VEL
LIN {X 0,Y 453.477,Z 343.625,A -85,B 0,C 180,E1 -8404.989,E2 -8404.989} C_VEL
LIN {X 0,Y 453.462,Z 343.627,A -85,B 0,C 180,E1 -8408.311,E2 -8408.311} C_VEL
LIN {X 0,Y 453.491,Z 343.617,A -85,B 0,C 180,E1 -8410.609,E2 -8410.609} C_VEL
LIN {X 0,Y 453.461,Z 343.629,A -85,B 0,C 180,E1 -8413.245,E2 -8413.245} C_VEL
LIN {X 0,Y 453.471,Z 343.621,A -85,B 0,C 180,E1 -8415.78,E2 -8415.78} C_VEL
LIN {X 0,Y 453.478,Z 343.618,A -85,B 0,C 180,E1 -8418.209,E2 -8418.209} C_VEL
LIN {X 0,Y 453.491,Z 343.62,A -85,B 0,C 180,E1 -8420.793,E2 -8420.793} C_VEL
LIN {X 0,Y 453.454,Z 343.622,A -85,B 0,C 180,E1 -8423.917,E2 -8423.917} C_VEL
LIN {X 0,Y 453.479,Z 343.626,A -85,B 0,C 180,E1 -8427.151,E2 -8427.151} C_VEL
LIN {X 0,Y 453.471,Z 343.619,A -85,B 0,C 180,E1 -8430.268,E2 -8430.268} C_VEL
LIN {X 0,Y 453.504,Z 343.62,A -85,B 0,C 180,E1 -8433.294,E2 -8433.294} C_VEL
LIN {X 0,Y 453.5,Z 343.616,A -85,B 0,C 180,E1 -8436.239,E2 -8436.239} C_VEL
LIN {X 0,Y 453.481,Z 343.625,A -85,B 0,C 180,E1 -8439.118,E2 -8439.118} C_VEL
LIN {X 0,Y 453.509,Z 343.614,A -85,B 0,C 180,E1 -8441.945,E2 -8441.945} C_VEL
LIN {X 0,Y 453.537,Z 343.615,A -85,B 0,C 180,E1 -8444.727,E2 -8444.727} C_VEL
LIN {X 0,Y 453.557,Z 343.61,A -85,B 0,C 180,E1 -8448.379,E2 -8448.379} C_VEL
LIN {X 0,Y 453.649,Z 343.597,A -85,B 0,C 180,E1 -8451.985,E2 -8451.985} C_VEL
LIN {X 0,Y 453.665,Z 343.599,A -85,B 0,C 180,E1 -8454.667,E2 -8454.667} C_VEL
LIN {X 0,Y 453.763,Z 343.586,A -85,B 0,C 180,E1 -8457.337,E2 -8457.337} C_VEL
LIN {X 0,Y 453.822,Z 343.575,A -85,B 0,C 180,E1 -8460,E2 -8460} C_VEL
LIN {X 0,Y 453.762,Z 343.588,A -85,B 0,C 180,E1 -8462.664,E2 -8462.664} C_VEL
LIN {X 0,Y 453.677,Z 343.594,A -85,B 0,C 180,E1 -8466.226,E2 -8466.226} C_VEL
LIN {X 0,Y 453.59,Z 343.611,A -85,B 0,C 180,E1 -8468.914,E2 -8468.914} C_VEL
LIN {X 0,Y 453.561,Z 343.612,A -85,B 0,C 180,E1 -8472.529,E2 -8472.529} C_VEL
LIN {X 0,Y 453.543,Z 343.611,A -85,B 0,C 180,E1 -8476.196,E2 -8476.196} C_VEL
LIN {X 0,Y 453.518,Z 343.618,A -85,B 0,C 180,E1 -8479.041,E2 -8479.041} C_VEL
LIN {X 0,Y 453.475,Z 343.619,A -85,B 0,C 180,E1 -8481.837,E2 -8481.837} C_VEL
LIN {X 0,Y 453.502,Z 343.624,A -85,B 0,C 180,E1 -8484.736,E2 -8484.736} C_VEL
LIN {X 0,Y 453.527,Z 343.613,A -85,B 0,C 180,E1 -8487.959,E2 -8487.959} C_VEL
LIN {X 0,Y 453.465,Z 343.62,A -85,B 0,C 180,E1 -8491.526,E2 -8491.526} C_VEL
LIN {X 0,Y 453.488,Z 343.623,A -85,B 0,C 180,E1 -8494.778,E2 -8494.778} C_VEL
LIN {X 0,Y 453.46,Z 343.624,A -85,B 0,C 180,E1 -8498.313,E2 -8498.313} C_VEL
LIN {X 0,Y 453.493,Z 343.625,A -85,B 0,C 180,E1 -8500.61,E2 -8500.61} C_VEL
LIN {X 0,Y 453.46,Z 343.624,A -85,B 0,C 180,E1 -8504.222,E2 -8504.222} C_VEL
LIN {X 0,Y 453.448,Z 343.624,A -85,B 0,C 180,E1 -8507.004,E2 -8507.004} C_VEL
LIN {X 0,Y 453.494,Z 343.616,A -85,B 0,C 180,E1 -8509.41,E2 -8509.41} C_VEL
LIN {X 0,Y 453.45,Z 343.626,A -85,B 0,C 180,E1 -8512.811,E2 -8512.811} C_VEL
LIN {X 0,Y 453.478,Z 343.621,A -85,B 0,C 180,E1 -8516.088,E2 -8516.088} C_VEL
LIN {X 0,Y 453.477,Z 343.619,A -85,B 0,C 180,E1 -8519.241,E2 -8519.241} C_VEL
LIN {X 0,Y 453.509,Z 343.62,A -85,B 0,C 180,E1 -8522.296,E2 -8522.296} C_VEL
LIN {X 0,Y 453.496,Z 343.616,A -85,B 0,C 180,E1 -8525.265,E2 -8525.265} C_VEL
LIN {X 0,Y 453.483,Z 343.626,A -85,B 0,C 180,E1 -8528.416,E2 -8528.416} C_VEL
LIN {X 0,Y 453.525,Z 343.613,A -85,B 0,C 180,E1 -8531.009,E2 -8531.009} C_VEL
LIN {X 0,Y 453.523,Z 343.616,A -85,B 0,C 180,E1 -8534.726,E2 -8534.726} C_VEL
LIN {X 0,Y 453.562,Z 343.616,A -85,B 0,C 180,E1 -8538.379,E2 -8538.379} C_VEL
LIN {X 0,Y 453.58,Z 343.606,A -85,B 0,C 180,E1 -8541.087,E2 -8541.087} C_VEL
LIN {X 0,Y 453.589,Z 343.605,A -85,B 0,C 180,E1 -8543.087,E2 -8543.087} C_VEL
LIN {X 0,Y 452.911,Z 343.693,A -85,B 0,C 180,E1 -8543.828,E2 -8543.828} C_VEL
LIN {X 0,Y 449.964,Z 344.058,A -85,B 0,C 180,E1 -8545.03,E2 -8545.03} C_VEL
LIN {X 0,Y 447.537,Z 344.362,A -85,B 0,C 180,E1 -8546,E2 -8546} C_VEL
LIN {X 0,Y 446.595,Z 344.479,A -85,B 0,C 180,E1 -8546.75,E2 -8546.75} C_VEL
LIN {X 0,Y 446.573,Z 344.479,A -85,B 0,C 180,E1 -8547.004,E2 -8547.004} C_VEL
LIN {X 0,Y 446.722,Z 344.464,A -85,B 0,C 180,E1 -8550,E2 -8550} C_VEL
LIN {X 0,Y 446.655,Z 344.471,A -85,B 0,C 180,E1 -8552.706,E2 -8552.706} C_VEL
LIN {X 0,Y 446.61,Z 344.481,A -85,B 0,C 180,E1 -8556.325,E2 -8556.325} C_VEL
LIN {X 0,Y 446.513,Z 344.486,A -85,B 0,C 180,E1 -8559.056,E2 -8559.056} C_VEL
LIN {X 0,Y 446.497,Z 344.49,A -85,B 0,C 180,E1 -8562.731,E2 -8562.731} C_VEL
LIN {X 0,Y 446.457,Z 344.617,A -85,B 0,C 180,E1 -8564.268,E2 -8564.268} C_VEL
LIN {X 0,Y 446.883,Z 346.363,A -85,B 0,C 180,E1 -8564.603,E2 -8564.603} C_VEL
LIN {X 0,Y 456.377,Z 369.106,A -85,B 0,C 180,E1 -8565.561,E2 -8565.561} C_VEL
LIN {X 0,Y 454.301,Z 510.847,A -85,B 0,C 180,E1 -8567.936,E2 -8567.936} C_VEL
LIN {X 0,Y 453.847,Z 526.581,A -85,B 0,C 180,E1 -8568.386,E2 -8568.386} C_VEL
LIN {X 0,Y 453.227,Z 541.595,A -85,B 0,C 180,E1 -8569.005,E2 -8569.005} C_VEL
LIN {X 0,Y 452.476,Z 555.329,A -85,B 0,C 180,E1 -8569.745,E2 -8569.745} C_VEL
LIN {X 0,Y 451.502,Z 569.907,A -85,B 0,C 180,E1 -8570.74,E2 -8570.74} C_VEL
LIN {X 0,Y 450.514,Z 583.218,A -85,B 0,C 180,E1 -8571.867,E2 -8571.867} C_VEL
LIN {X 0,Y 449.587,Z 595.451,A -85,B 0,C 180,E1 -8573.127,E2 -8573.127} C_VEL
LIN {X 0,Y 448.617,Z 607.059,A -85,B 0,C 180,E1 -8574.565,E2 -8574.565} C_VEL
LIN {X 0,Y 447.782,Z 617.173,A -85,B 0,C 180,E1 -8576.07,E2 -8576.07} C_VEL
LIN {X 0,Y 447.12,Z 625.906,A -85,B 0,C 180,E1 -8577.626,E2 -8577.626} C_VEL
LIN {X 0,Y 446.552,Z 633.257,A -85,B 0,C 180,E1 -8579.202,E2 -8579.202} C_VEL
LIN {X 0,Y 446.159,Z 639.393,A -85,B 0,C 180,E1 -8580.794,E2 -8580.794} C_VEL
LIN {X 0,Y 445.866,Z 644.475,A -85,B 0,C 180,E1 -8582.407,E2 -8582.407} C_VEL
LIN {X 0,Y 445.627,Z 648.566,A -85,B 0,C 180,E1 -8584.047,E2 -8584.047} C_VEL
LIN {X 0,Y 445.452,Z 651.605,A -85,B 0,C 180,E1 -8585.716,E2 -8585.716} C_VEL
LIN {X 0,Y 445.355,Z 653.127,A -85,B 0,C 180,E1 -8586.846,E2 -8586.846} C_VEL
LIN {X 0,Y 445.326,Z 654.208,A -85,B 0,C 180,E1 -8587.988,E2 -8587.988} C_VEL
LIN {X 0,Y 445.295,Z 654.855,A -85,B 0,C 180,E1 -8589.343,E2 -8589.343} C_VEL
LIN {X 0,Y 445.302,Z 654.885,A -85,B 0,C 180,E1 -8590.749,E2 -8590.749} C_VEL
LIN {X 0,Y 445.362,Z 653.767,A -85,B 0,C 180,E1 -8592.732,E2 -8592.732} C_VEL
LIN {X 0,Y 445.471,Z 652.405,A -85,B 0,C 180,E1 -8593.961,E2 -8593.961} C_VEL
LIN {X 0,Y 445.686,Z 648.781,A -85,B 0,C 180,E1 -8596.065,E2 -8596.065} C_VEL
LIN {X 0,Y 445.914,Z 644.511,A -85,B 0,C 180,E1 -8597.797,E2 -8597.797} C_VEL
LIN {X 0,Y 446.299,Z 638.126,A -85,B 0,C 180,E1 -8599.786,E2 -8599.786} C_VEL
LIN {X 0,Y 446.796,Z 631.316,A -85,B 0,C 180,E1 -8601.456,E2 -8601.456} C_VEL
LIN {X 0,Y 447.422,Z 623.581,A -85,B 0,C 180,E1 -8603.021,E2 -8603.021} C_VEL
LIN {X 0,Y 448.192,Z 614.061,A -85,B 0,C 180,E1 -8604.627,E2 -8604.627} C_VEL
LIN {X 0,Y 449.064,Z 603.981,A -85,B 0,C 180,E1 -8606.045,E2 -8606.045} C_VEL
LIN {X 0,Y 450.074,Z 592.326,A -85,B 0,C 180,E1 -8607.414,E2 -8607.414} C_VEL
LIN {X 0,Y 451.009,Z 579.84,A -85,B 0,C 180,E1 -8608.635,E2 -8608.635} C_VEL
LIN {X 0,Y 451.972,Z 567.3,A -85,B 0,C 180,E1 -8609.644,E2 -8609.644} C_VEL
LIN {X 0,Y 452.84,Z 553.154,A -85,B 0,C 180,E1 -8610.57,E2 -8610.57} C_VEL
LIN {X 0,Y 453.585,Z 539.057,A -85,B 0,C 180,E1 -8611.293,E2 -8611.293} C_VEL
LIN {X 0,Y 454.15,Z 523.373,A -85,B 0,C 180,E1 -8611.895,E2 -8611.895} C_VEL
LIN {X 0,Y 454.609,Z 508.326,A -85,B 0,C 180,E1 -8612.279,E2 -8612.279} C_VEL
LIN {X 0,Y 456.809,Z 369.768,A -85,B 0,C 180,E1 -8614.621,E2 -8614.621} C_VEL
LIN {X 0,Y 448.617,Z 350.88,A -85,B 0,C 180,E1 -8615.488,E2 -8615.488} C_VEL
LIN {X 0,Y 447.288,Z 347.937,A -85,B 0,C 180,E1 -8615.641,E2 -8615.641} C_VEL
LIN {X 0,Y 446.463,Z 344.501,A -85,B 0,C 180,E1 -8616.395,E2 -8616.395} C_VEL
LIN {X 0,Y 446.437,Z 344.504,A -85,B 0,C 180,E1 -8619.736,E2 -8619.736} C_VEL
LIN {X 0,Y 446.439,Z 344.495,A -85,B 0,C 180,E1 -8622.596,E2 -8622.596} C_VEL
LIN {X 0,Y 446.462,Z 344.499,A -85,B 0,C 180,E1 -8625.412,E2 -8625.412} C_VEL
LIN {X 0,Y 446.52,Z 344.49,A -85,B 0,C 180,E1 -8628.193,E2 -8628.193} C_VEL
LIN {X 0,Y 446.528,Z 344.487,A -85,B 0,C 180,E1 -8630.944,E2 -8630.944} C_VEL
LIN {X 0,Y 446.609,Z 344.481,A -85,B 0,C 180,E1 -8633.675,E2 -8633.675} C_VEL
LIN {X 0,Y 446.657,Z 344.472,A -85,B 0,C 180,E1 -8637.294,E2 -8637.294} C_VEL
LIN {X 0,Y 446.79,Z 344.456,A -85,B 0,C 180,E1 -8640,E2 -8640} C_VEL
LIN {X 0,Y 446.685,Z 344.466,A -85,B 0,C 180,E1 -8642.705,E2 -8642.705} C_VEL
LIN {X 0,Y 446.615,Z 344.475,A -85,B 0,C 180,E1 -8646.324,E2 -8646.324} C_VEL
LIN {X 0,Y 446.534,Z 344.489,A -85,B 0,C 180,E1 -8649.055,E2 -8649.055} C_VEL
LIN {X 0,Y 446.524,Z 344.486,A -85,B 0,C 180,E1 -8652.729,E2 -8652.729} C_VEL
LIN {X 0,Y 446.491,Z 344.488,A -85,B 0,C 180,E1 -8656.459,E2 -8656.459} C_VEL
LIN {X 0,Y 446.471,Z 344.495,A -85,B 0,C 180,E1 -8659.303,E2 -8659.303} C_VEL
LIN {X 0,Y 446.42,Z 344.498,A -85,B 0,C 180,E1 -8662.199,E2 -8662.199} C_VEL
LIN {X 0,Y 446.459,Z 344.497,A -85,B 0,C 180,E1 -8665.152,E2 -8665.152} C_VEL
LIN {X 0,Y 446.487,Z 344.491,A -85,B 0,C 180,E1 -8668.178,E2 -8668.178} C_VEL
LIN {X 0,Y 446.421,Z 344.499,A -85,B 0,C 180,E1 -8671.775,E2 -8671.775} C_VEL
LIN {X 0,Y 446.43,Z 344.501,A -85,B 0,C 180,E1 -8674.523,E2 -8674.523} C_VEL
LIN {X 0,Y 446.417,Z 344.502,A -85,B 0,C 180,E1 -8678.079,E2 -8678.079} C_VEL
LIN {X 0,Y 446.428,Z 344.503,A -85,B 0,C 180,E1 -8680.917,E2 -8680.917} C_VEL
LIN {X 0,Y 446.403,Z 344.503,A -85,B 0,C 180,E1 -8683.845,E2 -8683.845} C_VEL
LIN {X 0,Y 446.422,Z 344.502,A -85,B 0,C 180,E1 -8686.4,E2 -8686.4} C_VEL
LIN {X 0,Y 446.452,Z 344.499,A -85,B 0,C 180,E1 -8689.803,E2 -8689.803} C_VEL
LIN {X 0,Y 446.41,Z 344.505,A -85,B 0,C 180,E1 -8692.121,E2 -8692.121} C_VEL
LIN {X 0,Y 446.43,Z 344.502,A -85,B 0,C 180,E1 -8695.477,E2 -8695.477} C_VEL
LIN {X 0,Y 446.467,Z 344.552,A -85,B 0,C 180,E1 -8697.14,E2 -8697.14} C_VEL
LIN {X 0,Y 450.43,Z 359.944,A -85,B 0,C 180,E1 -8699.859,E2 -8699.859} C_VEL
LIN {X 0,Y 452.24,Z 367.927,A -85,B 0,C 180,E1 -8701.2,E2 -8701.2} C_VEL
LIN {X 0,Y 451.467,Z 381.319,A -85,B 0,C 180,E1 -8703.163,E2 -8703.163} C_VEL
LIN {X 0,Y 450.789,Z 391.369,A -85,B 0,C 180,E1 -8704.612,E2 -8704.612} C_VEL
LIN {X 0,Y 456.225,Z 421.956,A -85,B 0,C 180,E1 -8705.496,E2 -8705.496} C_VEL
LIN {X 0,Y 454.545,Z 534.567,A -85,B 0,C 180,E1 -8707.38,E2 -8707.38} C_VEL
LIN {X 0,Y 454.058,Z 560.254,A -85,B 0,C 180,E1 -8707.834,E2 -8707.834} C_VEL
LIN {X 0,Y 453.398,Z 575.987,A -85,B 0,C 180,E1 -8708.286,E2 -8708.286} C_VEL
LIN {X 0,Y 452.646,Z 590.399,A -85,B 0,C 180,E1 -8708.875,E2 -8708.875} C_VEL
LIN {X 0,Y 451.751,Z 604.539,A -85,B 0,C 180,E1 -8709.629,E2 -8709.629} C_VEL
LIN {X 0,Y 450.747,Z 618.017,A -85,B 0,C 180,E1 -8710.532,E2 -8710.532} C_VEL
LIN {X 0,Y 449.695,Z 631.782,A -85,B 0,C 180,E1 -8711.668,E2 -8711.668} C_VEL
LIN {X 0,Y 448.654,Z 644.779,A -85,B 0,C 180,E1 -8712.975,E2 -8712.975} C_VEL
LIN {X 0,Y 447.823,Z 655.727,A -85,B 0,C 180,E1 -8714.293,E2 -8714.293} C_VEL
LIN {X 0,Y 447.012,Z 666.846,A -85,B 0,C 180,E1 -8715.895,E2 -8715.895} C_VEL
LIN {X 0,Y 446.403,Z 675.829,A -85,B 0,C 180,E1 -8717.449,E2 -8717.449} C_VEL
LIN {X 0,Y 446.046,Z 683.775,A -85,B 0,C 180,E1 -8719.101,E2 -8719.101} C_VEL
LIN {X 0,Y 445.663,Z 690.953,A -85,B 0,C 180,E1 -8720.926,E2 -8720.926} C_VEL
LIN {X 0,Y 445.568,Z 696.616,A -85,B 0,C 180,E1 -8722.75,E2 -8722.75} C_VEL
LIN {X 0,Y 445.448,Z 700.901,A -85,B 0,C 180,E1 -8724.568,E2 -8724.568} C_VEL
LIN {X 0,Y 445.418,Z 703.916,A -85,B 0,C 180,E1 -8726.381,E2 -8726.381} C_VEL
LIN {X 0,Y 445.45,Z 705.726,A -85,B 0,C 180,E1 -8728.191,E2 -8728.191} C_VEL
LIN {X 0,Y 445.397,Z 706.36,A -85,B 0,C 180,E1 -8730,E2 -8730} C_VEL
LIN {X 0,Y 445.448,Z 705.775,A -85,B 0,C 180,E1 -8731.808,E2 -8731.808} C_VEL
LIN {X 0,Y 445.417,Z 704.008,A -85,B 0,C 180,E1 -8733.618,E2 -8733.618} C_VEL
LIN {X 0,Y 445.446,Z 701.041,A -85,B 0,C 180,E1 -8735.432,E2 -8735.432} C_VEL
LIN {X 0,Y 445.496,Z 696.802,A -85,B 0,C 180,E1 -8737.25,E2 -8737.25} C_VEL
LIN {X 0,Y 445.662,Z 691.182,A -85,B 0,C 180,E1 -8739.073,E2 -8739.073} C_VEL
LIN {X 0,Y 446.054,Z 684.034,A -85,B 0,C 180,E1 -8740.898,E2 -8740.898} C_VEL
LIN {X 0,Y 446.407,Z 676.095,A -85,B 0,C 180,E1 -8742.554,E2 -8742.554} C_VEL
LIN {X 0,Y 447.07,Z 667.169,A -85,B 0,C 180,E1 -8744.102,E2 -8744.102} C_VEL
LIN {X 0,Y 447.859,Z 656.042,A -85,B 0,C 180,E1 -8745.705,E2 -8745.705} C_VEL
LIN {X 0,Y 448.736,Z 644.773,A -85,B 0,C 180,E1 -8747.06,E2 -8747.06} C_VEL
LIN {X 0,Y 449.677,Z 632.069,A -85,B 0,C 180,E1 -8748.332,E2 -8748.332} C_VEL
LIN {X 0,Y 450.686,Z 619.744,A -85,B 0,C 180,E1 -8749.352,E2 -8749.352} C_VEL
LIN {X 0,Y 451.594,Z 606.434,A -85,B 0,C 180,E1 -8750.259,E2 -8750.259} C_VEL
LIN {X 0,Y 452.546,Z 592.395,A -85,B 0,C 180,E1 -8751.021,E2 -8751.021} C_VEL
LIN {X 0,Y 453.253,Z 577.513,A -85,B 0,C 180,E1 -8751.643,E2 -8751.643} C_VEL
LIN {X 0,Y 453.921,Z 562.459,A -85,B 0,C 180,E1 -8752.082,E2 -8752.082} C_VEL
LIN {X 0,Y 454.381,Z 538.847,A -85,B 0,C 180,E1 -8752.508,E2 -8752.508} C_VEL
LIN {X 0,Y 456.078,Z 422.412,A -85,B 0,C 180,E1 -8754.436,E2 -8754.436} C_VEL
LIN {X 0,Y 450.844,Z 392.86,A -85,B 0,C 180,E1 -8755.266,E2 -8755.266} C_VEL
LIN {X 0,Y 452.231,Z 371.771,A -85,B 0,C 180,E1 -8758.293,E2 -8758.293} C_VEL
LIN {X 0,Y 452.134,Z 367.316,A -85,B 0,C 180,E1 -8758.965,E2 -8758.965} C_VEL
LIN {X 0,Y 448.268,Z 351.598,A -85,B 0,C 180,E1 -8761.602,E2 -8761.602} C_VEL
LIN {X 0,Y 446.465,Z 344.497,A -85,B 0,C 180,E1 -8762.859,E2 -8762.859} C_VEL
LIN {X 0,Y 446.416,Z 344.503,A -85,B 0,C 180,E1 -8765.626,E2 -8765.626} C_VEL
LIN {X 0,Y 446.453,Z 344.503,A -85,B 0,C 180,E1 -8769.025,E2 -8769.025} C_VEL
LIN {X 0,Y 446.434,Z 344.496,A -85,B 0,C 180,E1 -8772.277,E2 -8772.277} C_VEL
LIN {X 0,Y 446.454,Z 344.5,A -85,B 0,C 180,E1 -8775.103,E2 -8775.103} C_VEL
LIN {X 0,Y 446.426,Z 344.498,A -85,B 0,C 180,E1 -8778.609,E2 -8778.609} C_VEL
LIN {X 0,Y 446.442,Z 344.5,A -85,B 0,C 180,E1 -8780.973,E2 -8780.973} C_VEL
LIN {X 0,Y 446.418,Z 344.498,A -85,B 0,C 180,E1 -8784.374,E2 -8784.374} C_VEL
LIN {X 0,Y 446.419,Z 344.5,A -85,B 0,C 180,E1 -8787.638,E2 -8787.638} C_VEL
LIN {X 0,Y 446.445,Z 344.498,A -85,B 0,C 180,E1 -8790.791,E2 -8790.791} C_VEL
LIN {X 0,Y 446.474,Z 344.491,A -85,B 0,C 180,E1 -8793.848,E2 -8793.848} C_VEL
LIN {X 0,Y 446.426,Z 344.501,A -85,B 0,C 180,E1 -8796.823,E2 -8796.823} C_VEL
LIN {X 0,Y 446.442,Z 344.495,A -85,B 0,C 180,E1 -8799.737,E2 -8799.737} C_VEL
LIN {X 0,Y 446.461,Z 344.495,A -85,B 0,C 180,E1 -8802.597,E2 -8802.597} C_VEL
LIN {X 0,Y 446.468,Z 344.494,A -85,B 0,C 180,E1 -8805.413,E2 -8805.413} C_VEL
LIN {X 0,Y 446.515,Z 344.486,A -85,B 0,C 180,E1 -8808.193,E2 -8808.193} C_VEL
LIN {X 0,Y 446.597,Z 344.475,A -85,B 0,C 180,E1 -8811.858,E2 -8811.858} C_VEL
LIN {X 0,Y 446.639,Z 344.473,A -85,B 0,C 180,E1 -8814.583,E2 -8814.583} C_VEL
LIN {X 0,Y 446.707,Z 344.465,A -85,B 0,C 180,E1 -8817.295,E2 -8817.295} C_VEL
LIN {X 0,Y 446.792,Z 344.451,A -85,B 0,C 180,E1 -8820,E2 -8820} C_VEL
LIN {X 0,Y 446.706,Z 344.467,A -85,B 0,C 180,E1 -8822.706,E2 -8822.706} C_VEL
LIN {X 0,Y 446.646,Z 344.471,A -85,B 0,C 180,E1 -8826.324,E2 -8826.324} C_VEL
LIN {X 0,Y 446.536,Z 344.488,A -85,B 0,C 180,E1 -8829.056,E2 -8829.056} C_VEL
LIN {X 0,Y 446.519,Z 344.492,A -85,B 0,C 180,E1 -8832.73,E2 -8832.73} C_VEL
LIN {X 0,Y 446.494,Z 344.49,A -85,B 0,C 180,E1 -8836.228,E2 -8836.228} C_VEL
LIN {X 0,Y 446.468,Z 344.493,A -85,B 0,C 180,E1 -8839.304,E2 -8839.304} C_VEL
LIN {X 0,Y 446.416,Z 344.5,A -85,B 0,C 180,E1 -8842.2,E2 -8842.2} C_VEL
LIN {X 0,Y 446.442,Z 344.497,A -85,B 0,C 180,E1 -8845.154,E2 -8845.154} C_VEL
LIN {X 0,Y 446.483,Z 344.491,A -85,B 0,C 180,E1 -8848.179,E2 -8848.179} C_VEL
LIN {X 0,Y 446.418,Z 344.498,A -85,B 0,C 180,E1 -8851.775,E2 -8851.775} C_VEL
LIN {X 0,Y 446.43,Z 344.502,A -85,B 0,C 180,E1 -8854.523,E2 -8854.523} C_VEL
LIN {X 0,Y 446.413,Z 344.5,A -85,B 0,C 180,E1 -8858.08,E2 -8858.08} C_VEL
LIN {X 0,Y 446.421,Z 344.501,A -85,B 0,C 180,E1 -8860.917,E2 -8860.917} C_VEL
LIN {X 0,Y 446.398,Z 344.501,A -85,B 0,C 180,E1 -8863.847,E2 -8863.847} C_VEL
LIN {X 0,Y 446.398,Z 344.506,A -85,B 0,C 180,E1 -8866.404,E2 -8866.404} C_VEL
LIN {X 0,Y 446.441,Z 344.495,A -85,B 0,C 180,E1 -8869.802,E2 -8869.802} C_VEL
LIN {X 0,Y 446.401,Z 344.5,A -85,B 0,C 180,E1 -8873.255,E2 -8873.255} C_VEL
LIN {X 0,Y 446.45,Z 344.501,A -85,B 0,C 180,E1 -8876.567,E2 -8876.567} C_VEL
LIN {X 0,Y 446.43,Z 344.498,A -85,B 0,C 180,E1 -8879.98,E2 -8879.98} C_VEL
LIN {X 0,Y 446.446,Z 344.497,A -85,B 0,C 180,E1 -8882.838,E2 -8882.838} C_VEL
LIN {X 0,Y 446.463,Z 344.494,A -85,B 0,C 180,E1 -8885.926,E2 -8885.926} C_VEL
LIN {X 0,Y 446.456,Z 344.496,A -85,B 0,C 180,E1 -8888.774,E2 -8888.774} C_VEL
LIN {X 0,Y 446.443,Z 344.495,A -85,B 0,C 180,E1 -8891.649,E2 -8891.649} C_VEL
LIN {X 0,Y 446.463,Z 344.499,A -85,B 0,C 180,E1 -8894.479,E2 -8894.479} C_VEL
LIN {X 0,Y 446.52,Z 344.485,A -85,B 0,C 180,E1 -8897.384,E2 -8897.384} C_VEL
LIN {X 0,Y 446.529,Z 344.485,A -85,B 0,C 180,E1 -8900.945,E2 -8900.945} C_VEL
LIN {X 0,Y 446.609,Z 344.475,A -85,B 0,C 180,E1 -8903.676,E2 -8903.676} C_VEL
LIN {X 0,Y 446.573,Z 344.479,A -85,B 0,C 180,E1 -8907.004,E2 -8907.004} C_VEL
LIN {X 0,Y 446.364,Z 344.506,A -85,B 0,C 180,E1 -8907.507,E2 -8907.507} C_VEL
LIN {X 0,Y 445.081,Z 344.672,A -85,B 0,C 180,E1 -8908.25,E2 -8908.25} C_VEL
LIN {X 0,Y 440.698,Z 345.214,A -85,B 0,C 180,E1 -8909.965,E2 -8909.965} C_VEL
LIN {X 0,Y 439.633,Z 345.346,A -85,B 0,C 180,E1 -8910.728,E2 -8910.728} C_VEL
LIN {X 0,Y 439.555,Z 345.353,A -85,B 0,C 180,E1 -8910.987,E2 -8910.987} C_VEL
LIN {X 0,Y 439.606,Z 345.348,A -85,B 0,C 180,E1 -8912.749,E2 -8912.749} C_VEL
LIN {X 0,Y 439.563,Z 345.358,A -85,B 0,C 180,E1 -8916.426,E2 -8916.426} C_VEL
LIN {X 0,Y 439.479,Z 345.362,A -85,B 0,C 180,E1 -8919.202,E2 -8919.202} C_VEL
LIN {X 0,Y 439.456,Z 345.367,A -85,B 0,C 180,E1 -8922.938,E2 -8922.938} C_VEL
LIN {X 0,Y 439.422,Z 345.492,A -85,B 0,C 180,E1 -8923.94,E2 -8923.94} C_VEL
LIN {X 0,Y 439.763,Z 346.877,A -85,B 0,C 180,E1 -8924.18,E2 -8924.18} C_VEL
LIN {X 0,Y 449.922,Z 370.988,A -85,B 0,C 180,E1 -8925.226,E2 -8925.226} C_VEL
LIN {X 0,Y 447.704,Z 511.543,A -85,B 0,C 180,E1 -8927.619,E2 -8927.619} C_VEL
LIN {X 0,Y 447.23,Z 526.577,A -85,B 0,C 180,E1 -8928.052,E2 -8928.052} C_VEL
LIN {X 0,Y 446.612,Z 541.63,A -85,B 0,C 180,E1 -8928.677,E2 -8928.677} C_VEL
LIN {X 0,Y 445.781,Z 555.886,A -85,B 0,C 180,E1 -8929.454,E2 -8929.454} C_VEL
LIN {X 0,Y 444.806,Z 570.073,A -85,B 0,C 180,E1 -8930.436,E2 -8930.436} C_VEL
LIN {X 0,Y 443.723,Z 583.727,A -85,B 0,C 180,E1 -8931.608,E2 -8931.608} C_VEL
LIN {X 0,Y 442.794,Z 595.639,A -85,B 0,C 180,E1 -8932.851,E2 -8932.851} C_VEL
LIN {X 0,Y 441.825,Z 606.347,A -85,B 0,C 180,E1 -8934.18,E2 -8934.18} C_VEL
LIN {X 0,Y 440.913,Z 616.873,A -85,B 0,C 180,E1 -8935.745,E2 -8935.745} C_VEL
LIN {X 0,Y 440.2,Z 625.775,A -85,B 0,C 180,E1 -8937.34,E2 -8937.34} C_VEL
LIN {X 0,Y 439.524,Z 634.289,A -85,B 0,C 180,E1 -8939.19,E2 -8939.19} C_VEL
LIN {X 0,Y 439.114,Z 640.313,A -85,B 0,C 180,E1 -8940.808,E2 -8940.808} C_VEL
LIN {X 0,Y 438.794,Z 645.284,A -85,B 0,C 180,E1 -8942.449,E2 -8942.449} C_VEL
LIN {X 0,Y 438.531,Z 649.282,A -85,B 0,C 180,E1 -8944.12,E2 -8944.12} C_VEL
LIN {X 0,Y 438.416,Z 651.363,A -85,B 0,C 180,E1 -8945.247,E2 -8945.247} C_VEL
LIN {X 0,Y 438.281,Z 653.403,A -85,B 0,C 180,E1 -8946.7,E2 -8946.7} C_VEL
LIN {X 0,Y 438.208,Z 655.036,A -85,B 0,C 180,E1 -8948.718,E2 -8948.718} C_VEL
LIN {X 0,Y 438.202,Z 655.375,A -85,B 0,C 180,E1 -8949.907,E2 -8949.907} C_VEL
LIN {X 0,Y 438.228,Z 655.233,A -85,B 0,C 180,E1 -8951.112,E2 -8951.112} C_VEL
LIN {X 0,Y 438.269,Z 654.443,A -85,B 0,C 180,E1 -8952.468,E2 -8952.468} C_VEL
LIN {X 0,Y 438.365,Z 653.065,A -85,B 0,C 180,E1 -8953.825,E2 -8953.825} C_VEL
LIN {X 0,Y 438.509,Z 651.125,A -85,B 0,C 180,E1 -8955.154,E2 -8955.154} C_VEL
LIN {X 0,Y 438.777,Z 647.32,A -85,B 0,C 180,E1 -8956.998,E2 -8956.998} C_VEL
LIN {X 0,Y 439.042,Z 641.822,A -85,B 0,C 180,E1 -8958.98,E2 -8958.98} C_VEL
LIN {X 0,Y 439.548,Z 635.164,A -85,B 0,C 180,E1 -8960.833,E2 -8960.833} C_VEL
LIN {X 0,Y 440.241,Z 627.016,A -85,B 0,C 180,E1 -8962.653,E2 -8962.653} C_VEL
LIN {X 0,Y 441.056,Z 617.681,A -85,B 0,C 180,E1 -8964.357,E2 -8964.357} C_VEL
LIN {X 0,Y 442.031,Z 606.763,A -85,B 0,C 180,E1 -8965.995,E2 -8965.995} C_VEL
LIN {X 0,Y 443.079,Z 595.763,A -85,B 0,C 180,E1 -8967.364,E2 -8967.364} C_VEL
LIN {X 0,Y 444.096,Z 582.7,A -85,B 0,C 180,E1 -8968.713,E2 -8968.713} C_VEL
LIN {X 0,Y 445.124,Z 569.83,A -85,B 0,C 180,E1 -8969.802,E2 -8969.802} C_VEL
LIN {X 0,Y 446.115,Z 555.735,A -85,B 0,C 180,E1 -8970.766,E2 -8970.766} C_VEL
LIN {X 0,Y 446.852,Z 542.566,A -85,B 0,C 180,E1 -8971.487,E2 -8971.487} C_VEL
LIN {X 0,Y 447.511,Z 527.076,A -85,B 0,C 180,E1 -8972.13,E2 -8972.13} C_VEL
LIN {X 0,Y 448.023,Z 511.984,A -85,B 0,C 180,E1 -8972.561,E2 -8972.561} C_VEL
LIN {X 0,Y 450.395,Z 371.595,A -85,B 0,C 180,E1 -8974.99,E2 -8974.99} C_VEL
LIN {X 0,Y 443.122,Z 354.783,A -85,B 0,C 180,E1 -8975.777,E2 -8975.777} C_VEL
LIN {X 0,Y 440.172,Z 348.429,A -85,B 0,C 180,E1 -8976.118,E2 -8976.118} C_VEL
LIN {X 0,Y 439.388,Z 345.379,A -85,B 0,C 180,E1 -8976.804,E2 -8976.804} C_VEL
LIN {X 0,Y 439.382,Z 345.378,A -85,B 0,C 180,E1 -8979.396,E2 -8979.396} C_VEL
LIN {X 0,Y 439.393,Z 345.374,A -85,B 0,C 180,E1 -8982.308,E2 -8982.308} C_VEL
LIN {X 0,Y 439.406,Z 345.376,A -85,B 0,C 180,E1 -8985.172,E2 -8985.172} C_VEL
LIN {X 0,Y 439.486,Z 345.368,A -85,B 0,C 180,E1 -8988.001,E2 -8988.001} C_VEL
LIN {X 0,Y 439.504,Z 345.366,A -85,B 0,C 180,E1 -8991.725,E2 -8991.725} C_VEL
LIN {X 0,Y 439.601,Z 345.349,A -85,B 0,C 180,E1 -8994.495,E2 -8994.495} C_VEL
LIN {X 0,Y 439.629,Z 345.347,A -85,B 0,C 180,E1 -8998.167,E2 -8998.167} C_VEL
LIN {X 0,Y 439.759,Z 345.332,A -85,B 0,C 180,E1 -9000,E2 -9000} C_VEL
LIN {X 0,Y 439.634,Z 345.344,A -85,B 0,C 180,E1 -9002.749,E2 -9002.749} C_VEL
LIN {X 0,Y 439.567,Z 345.353,A -85,B 0,C 180,E1 -9006.426,E2 -9006.426} C_VEL
LIN {X 0,Y 439.497,Z 345.367,A -85,B 0,C 180,E1 -9009.201,E2 -9009.201} C_VEL
LIN {X 0,Y 439.468,Z 345.365,A -85,B 0,C 180,E1 -9012.937,E2 -9012.937} C_VEL
LIN {X 0,Y 439.449,Z 345.365,A -85,B 0,C 180,E1 -9016.348,E2 -9016.348} C_VEL
LIN {X 0,Y 439.404,Z 345.376,A -85,B 0,C 180,E1 -9019.626,E2 -9019.626} C_VEL
LIN {X 0,Y 439.367,Z 345.378,A -85,B 0,C 180,E1 -9022.575,E2 -9022.575} C_VEL
LIN {X 0,Y 439.407,Z 345.376,A -85,B 0,C 180,E1 -9025.584,E2 -9025.584} C_VEL
LIN {X 0,Y 439.419,Z 345.374,A -85,B 0,C 180,E1 -9028.673,E2 -9028.673} C_VEL
LIN {X 0,Y 439.372,Z 345.376,A -85,B 0,C 180,E1 -9032.03,E2 -9032.03} C_VEL
LIN {X 0,Y 439.396,Z 345.38,A -85,B 0,C 180,E1 -9035.34,E2 -9035.34} C_VEL
LIN {X 0,Y 439.385,Z 345.381,A -85,B 0,C 180,E1 -9038.595,E2 -9038.595} C_VEL
LIN {X 0,Y 439.39,Z 345.379,A -85,B 0,C 180,E1 -9041.256,E2 -9041.256} C_VEL
LIN {X 0,Y 439.404,Z 345.377,A -85,B 0,C 180,E1 -9044.729,E2 -9044.729} C_VEL
LIN {X 0,Y 439.399,Z 345.376,A -85,B 0,C 180,E1 -9047.796,E2 -9047.796} C_VEL
LIN {X 0,Y 439.438,Z 345.374,A -85,B 0,C 180,E1 -9050.228,E2 -9050.228} C_VEL
LIN {X 0,Y 439.376,Z 345.379,A -85,B 0,C 180,E1 -9053.713,E2 -9053.713} C_VEL
LIN {X 0,Y 439.431,Z 345.512,A -85,B 0,C 180,E1 -9056.736,E2 -9056.736} C_VEL
LIN {X 0,Y 443.483,Z 360.898,A -85,B 0,C 180,E1 -9059.528,E2 -9059.528} C_VEL
LIN {X 0,Y 445.345,Z 369.314,A -85,B 0,C 180,E1 -9060.97,E2 -9060.97} C_VEL
LIN {X 0,Y 445.306,Z 374.317,A -85,B 0,C 180,E1 -9061.74,E2 -9061.74} C_VEL
LIN {X 0,Y 444.08,Z 390.819,A -85,B 0,C 180,E1 -9064.168,E2 -9064.168} C_VEL
LIN {X 0,Y 449.591,Z 421.47,A -85,B 0,C 180,E1 -9065.091,E2 -9065.091} C_VEL
LIN {X 0,Y 449.852,Z 425.145,A -85,B 0,C 180,E1 -9065.174,E2 -9065.174} C_VEL
LIN {X 0,Y 447.572,Z 558.871,A -85,B 0,C 180,E1 -9067.465,E2 -9067.465} C_VEL
LIN {X 0,Y 446.87,Z 574.637,A -85,B 0,C 180,E1 -9067.912,E2 -9067.912} C_VEL
LIN {X 0,Y 446.071,Z 588.81,A -85,B 0,C 180,E1 -9068.485,E2 -9068.485} C_VEL
LIN {X 0,Y 445.202,Z 602.202,A -85,B 0,C 180,E1 -9069.195,E2 -9069.195} C_VEL
LIN {X 0,Y 444.133,Z 616.035,A -85,B 0,C 180,E1 -9070.109,E2 -9070.109} C_VEL
LIN {X 0,Y 443.069,Z 628.772,A -85,B 0,C 180,E1 -9071.144,E2 -9071.144} C_VEL
LIN {X 0,Y 442.112,Z 640.625,A -85,B 0,C 180,E1 -9072.3,E2 -9072.3} C_VEL
LIN {X 0,Y 441.228,Z 651.659,A -85,B 0,C 180,E1 -9073.577,E2 -9073.577} C_VEL
LIN {X 0,Y 440.384,Z 661.874,A -85,B 0,C 180,E1 -9074.969,E2 -9074.969} C_VEL
LIN {X 0,Y 439.668,Z 671.881,A -85,B 0,C 180,E1 -9076.598,E2 -9076.598} C_VEL
LIN {X 0,Y 439.125,Z 680.239,A -85,B 0,C 180,E1 -9078.225,E2 -9078.225} C_VEL
LIN {X 0,Y 438.719,Z 687.143,A -85,B 0,C 180,E1 -9079.85,E2 -9079.85} C_VEL
LIN {X 0,Y 438.529,Z 693.548,A -85,B 0,C 180,E1 -9081.707,E2 -9081.707} C_VEL
LIN {X 0,Y 438.4,Z 698.803,A -85,B 0,C 180,E1 -9083.679,E2 -9083.679} C_VEL
LIN {X 0,Y 438.31,Z 702.149,A -85,B 0,C 180,E1 -9085.401,E2 -9085.401} C_VEL
LIN {X 0,Y 438.399,Z 704.562,A -85,B 0,C 180,E1 -9087.243,E2 -9087.243} C_VEL
LIN {X 0,Y 438.363,Z 705.781,A -85,B 0,C 180,E1 -9089.081,E2 -9089.081} C_VEL
LIN {X 0,Y 438.362,Z 705.81,A -85,B 0,C 180,E1 -9090.918,E2 -9090.918} C_VEL
LIN {X 0,Y 438.391,Z 704.629,A -85,B 0,C 180,E1 -9092.756,E2 -9092.756} C_VEL
LIN {X 0,Y 438.308,Z 702.258,A -85,B 0,C 180,E1 -9094.598,E2 -9094.598} C_VEL
LIN {X 0,Y 438.362,Z 698.658,A -85,B 0,C 180,E1 -9096.443,E2 -9096.443} C_VEL
LIN {X 0,Y 438.528,Z 693.737,A -85,B 0,C 180,E1 -9098.293,E2 -9098.293} C_VEL
LIN {X 0,Y 438.72,Z 687.354,A -85,B 0,C 180,E1 -9100.149,E2 -9100.149} C_VEL
LIN {X 0,Y 439.148,Z 680.48,A -85,B 0,C 180,E1 -9101.773,E2 -9101.773} C_VEL
LIN {X 0,Y 439.7,Z 672.152,A -85,B 0,C 180,E1 -9103.4,E2 -9103.4} C_VEL
LIN {X 0,Y 440.415,Z 662.153,A -85,B 0,C 180,E1 -9105.029,E2 -9105.029} C_VEL
LIN {X 0,Y 441.27,Z 651.916,A -85,B 0,C 180,E1 -9106.421,E2 -9106.421} C_VEL
LIN {X 0,Y 442.211,Z 639.75,A -85,B 0,C 180,E1 -9107.814,E2 -9107.814} C_VEL
LIN {X 0,Y 443.175,Z 627.583,A -85,B 0,C 180,E1 -9108.971,E2 -9108.971} C_VEL
LIN {X 0,Y 444.219,Z 614.399,A -85,B 0,C 180,E1 -9110.006,E2 -9110.006} C_VEL
LIN {X 0,Y 445.169,Z 601.934,A -85,B 0,C 180,E1 -9110.806,E2 -9110.806} C_VEL
LIN {X 0,Y 446.126,Z 586.887,A -85,B 0,C 180,E1 -9111.572,E2 -9111.572} C_VEL
LIN {X 0,Y 446.887,Z 571.518,A -85,B 0,C 180,E1 -9112.151,E2 -9112.151} C_VEL
LIN {X 0,Y 447.431,Z 556.111,A -85,B 0,C 180,E1 -9112.541,E2 -9112.541} C_VEL
LIN {X 0,Y 449.395,Z 436.089,A -85,B 0,C 180,E1 -9114.562,E2 -9114.562} C_VEL
LIN {X 0,Y 449.399,Z 422.042,A -85,B 0,C 180,E1 -9114.812,E2 -9114.812} C_VEL
LIN {X 0,Y 444.05,Z 392.412,A -85,B 0,C 180,E1 -9115.674,E2 -9115.674} C_VEL
LIN {X 0,Y 445.464,Z 373.001,A -85,B 0,C 180,E1 -9118.505,E2 -9118.505} C_VEL
LIN {X 0,Y 445.418,Z 369.604,A -85,B 0,C 180,E1 -9119.024,E2 -9119.024} C_VEL
LIN {X 0,Y 441.99,Z 355.319,A -85,B 0,C 180,E1 -9121.446,E2 -9121.446} C_VEL
LIN {X 0,Y 439.412,Z 345.378,A -85,B 0,C 180,E1 -9123.232,E2 -9123.232} C_VEL
LIN {X 0,Y 439.371,Z 345.381,A -85,B 0,C 180,E1 -9126.287,E2 -9126.287} C_VEL
LIN {X 0,Y 439.403,Z 345.373,A -85,B 0,C 180,E1 -9129.85,E2 -9129.85} C_VEL
LIN {X 0,Y 439.383,Z 345.375,A -85,B 0,C 180,E1 -9132.627,E2 -9132.627} C_VEL
LIN {X 0,Y 439.403,Z 345.379,A -85,B 0,C 180,E1 -9135.271,E2 -9135.271} C_VEL
LIN {X 0,Y 439.386,Z 345.376,A -85,B 0,C 180,E1 -9138.743,E2 -9138.743} C_VEL
LIN {X 0,Y 439.379,Z 345.377,A -85,B 0,C 180,E1 -9141.606,E2 -9141.606} C_VEL
LIN {X 0,Y 439.398,Z 345.376,A -85,B 0,C 180,E1 -9144.844,E2 -9144.844} C_VEL
LIN {X 0,Y 439.369,Z 345.376,A -85,B 0,C 180,E1 -9148.14,E2 -9148.14} C_VEL
LIN {X 0,Y 439.429,Z 345.37,A -85,B 0,C 180,E1 -9151.598,E2 -9151.598} C_VEL
LIN {X 0,Y 439.402,Z 345.373,A -85,B 0,C 180,E1 -9154.415,E2 -9154.415} C_VEL
LIN {X 0,Y 439.362,Z 345.38,A -85,B 0,C 180,E1 -9157.425,E2 -9157.425} C_VEL
LIN {X 0,Y 439.438,Z 345.37,A -85,B 0,C 180,E1 -9160.663,E2 -9160.663} C_VEL
LIN {X 0,Y 439.459,Z 345.365,A -85,B 0,C 180,E1 -9164.225,E2 -9164.225} C_VEL
LIN {X 0,Y 439.481,Z 345.362,A -85,B 0,C 180,E1 -9168.002,E2 -9168.002} C_VEL
LIN {X 0,Y 439.545,Z 345.354,A -85,B 0,C 180,E1 -9171.727,E2 -9171.727} C_VEL
LIN {X 0,Y 439.615,Z 345.348,A -85,B 0,C 180,E1 -9174.496,E2 -9174.496} C_VEL
LIN {X 0,Y 439.633,Z 345.343,A -85,B 0,C 180,E1 -9178.168,E2 -9178.168} C_VEL
LIN {X 0,Y 439.762,Z 345.327,A -85,B 0,C 180,E1 -9180,E2 -9180} C_VEL
LIN {X 0,Y 439.652,Z 345.347,A -85,B 0,C 180,E1 -9182.749,E2 -9182.749} C_VEL
LIN {X 0,Y 439.618,Z 345.347,A -85,B 0,C 180,E1 -9186.426,E2 -9186.426} C_VEL
LIN {X 0,Y 439.498,Z 345.363,A -85,B 0,C 180,E1 -9189.202,E2 -9189.202} C_VEL
LIN {X 0,Y 439.463,Z 345.37,A -85,B 0,C 180,E1 -9192.938,E2 -9192.938} C_VEL
LIN {X 0,Y 439.445,Z 345.369,A -85,B 0,C 180,E1 -9196.349,E2 -9196.349} C_VEL
LIN {X 0,Y 439.401,Z 345.372,A -85,B 0,C 180,E1 -9199.627,E2 -9199.627} C_VEL
LIN {X 0,Y 439.363,Z 345.382,A -85,B 0,C 180,E1 -9202.576,E2 -9202.576} C_VEL
LIN {X 0,Y 439.388,Z 345.374,A -85,B 0,C 180,E1 -9205.586,E2 -9205.586} C_VEL
LIN {X 0,Y 439.416,Z 345.378,A -85,B 0,C 180,E1 -9208.674,E2 -9208.674} C_VEL
LIN {X 0,Y 439.369,Z 345.377,A -85,B 0,C 180,E1 -9212.031,E2 -9212.031} C_VEL
LIN {X 0,Y 439.395,Z 345.373,A -85,B 0,C 180,E1 -9215.341,E2 -9215.341} C_VEL
LIN {X 0,Y 439.37,Z 345.383,A -85,B 0,C 180,E1 -9218.597,E2 -9218.597} C_VEL
LIN {X 0,Y 439.381,Z 345.375,A -85,B 0,C 180,E1 -9221.256,E2 -9221.256} C_VEL
LIN {X 0,Y 439.398,Z 345.378,A -85,B 0,C 180,E1 -9224.73,E2 -9224.73} C_VEL
LIN {X 0,Y 439.384,Z 345.374,A -85,B 0,C 180,E1 -9227.795,E2 -9227.795} C_VEL
LIN {X 0,Y 439.393,Z 345.377,A -85,B 0,C 180,E1 -9230.224,E2 -9230.224} C_VEL
LIN {X 0,Y 439.373,Z 345.376,A -85,B 0,C 180,E1 -9233.713,E2 -9233.713} C_VEL
LIN {X 0,Y 439.374,Z 345.377,A -85,B 0,C 180,E1 -9237.055,E2 -9237.055} C_VEL
LIN {X 0,Y 439.379,Z 345.38,A -85,B 0,C 180,E1 -9240.274,E2 -9240.274} C_VEL
LIN {X 0,Y 439.383,Z 345.374,A -85,B 0,C 180,E1 -9243.394,E2 -9243.394} C_VEL
LIN {X 0,Y 439.385,Z 345.382,A -85,B 0,C 180,E1 -9246.43,E2 -9246.43} C_VEL
LIN {X 0,Y 439.39,Z 345.373,A -85,B 0,C 180,E1 -9249.398,E2 -9249.398} C_VEL
LIN {X 0,Y 439.393,Z 345.38,A -85,B 0,C 180,E1 -9252.308,E2 -9252.308} C_VEL
LIN {X 0,Y 439.405,Z 345.372,A -85,B 0,C 180,E1 -9255.173,E2 -9255.173} C_VEL
LIN {X 0,Y 439.487,Z 345.365,A -85,B 0,C 180,E1 -9258.002,E2 -9258.002} C_VEL
LIN {X 0,Y 439.505,Z 345.36,A -85,B 0,C 180,E1 -9261.726,E2 -9261.726} C_VEL
LIN {X 0,Y 439.6,Z 345.352,A -85,B 0,C 180,E1 -9264.496,E2 -9264.496} C_VEL
LIN {X 0,Y 439.631,Z 345.35,A -85,B 0,C 180,E1 -9268.168,E2 -9268.168} C_VEL
LIN {X 0,Y 439.673,Z 345.342,A -85,B 0,C 180,E1 -9270,E2 -9270} C_VEL
LIN {X 0,Y 439.555,Z 345.353,A -85,B 0,C 180,E1 -9270.987,E2 -9270.987} C_VEL
LIN {X 0,Y 438.88,Z 345.44,A -85,B 0,C 180,E1 -9271.751,E2 -9271.751} C_VEL
LIN {X 0,Y 435.924,Z 345.806,A -85,B 0,C 180,E1 -9272.99,E2 -9272.99} C_VEL
LIN {X 0,Y 433.463,Z 346.116,A -85,B 0,C 180,E1 -9273.991,E2 -9273.991} C_VEL
LIN {X 0,Y 432.475,Z 346.237,A -85,B 0,C 180,E1 -9274.766,E2 -9274.766} C_VEL
LIN {X 0,Y 432.433,Z 346.24,A -85,B 0,C 180,E1 -9275.028,E2 -9275.028} C_VEL
LIN {X 0,Y 432.518,Z 346.23,A -85,B 0,C 180,E1 -9277.607,E2 -9277.607} C_VEL
LIN {X 0,Y 432.376,Z 346.249,A -85,B 0,C 180,E1 -9281.248,E2 -9281.248} C_VEL
LIN {X 0,Y 432.391,Z 346.374,A -85,B 0,C 180,E1 -9283.602,E2 -9283.602} C_VEL
LIN {X 0,Y 432.554,Z 347.137,A -85,B 0,C 180,E1 -9283.734,E2 -9283.734} C_VEL
LIN {X 0,Y 443.383,Z 372.675,A -85,B 0,C 180,E1 -9284.875,E2 -9284.875} C_VEL
LIN {X 0,Y 441.12,Z 511.858,A -85,B 0,C 180,E1 -9287.286,E2 -9287.286} C_VEL
LIN {X 0,Y 440.62,Z 527.058,A -85,B 0,C 180,E1 -9287.731,E2 -9287.731} C_VEL
LIN {X 0,Y 439.971,Z 541.4,A -85,B 0,C 180,E1 -9288.33,E2 -9288.33} C_VEL
LIN {X 0,Y 439.166,Z 554.923,A -85,B 0,C 180,E1 -9289.069,E2 -9289.069} C_VEL
LIN {X 0,Y 438.178,Z 569.214,A -85,B 0,C 180,E1 -9290.05,E2 -9290.05} C_VEL
LIN {X 0,Y 437.08,Z 582.237,A -85,B 0,C 180,E1 -9291.154,E2 -9291.154} C_VEL
LIN {X 0,Y 436.094,Z 594.144,A -85,B 0,C 180,E1 -9292.38,E2 -9292.38} C_VEL
LIN {X 0,Y 435.018,Z 605.847,A -85,B 0,C 180,E1 -9293.822,E2 -9293.822} C_VEL
LIN {X 0,Y 434.051,Z 616.645,A -85,B 0,C 180,E1 -9295.429,E2 -9295.429} C_VEL
LIN {X 0,Y 433.306,Z 625.454,A -85,B 0,C 180,E1 -9297.01,E2 -9297.01} C_VEL
LIN {X 0,Y 432.608,Z 633.238,A -85,B 0,C 180,E1 -9298.685,E2 -9298.685} C_VEL
LIN {X 0,Y 432.115,Z 639.985,A -85,B 0,C 180,E1 -9300.457,E2 -9300.457} C_VEL
LIN {X 0,Y 431.774,Z 645.26,A -85,B 0,C 180,E1 -9302.176,E2 -9302.176} C_VEL
LIN {X 0,Y 431.508,Z 649.286,A -85,B 0,C 180,E1 -9303.835,E2 -9303.835} C_VEL
LIN {X 0,Y 431.255,Z 652.918,A -85,B 0,C 180,E1 -9305.922,E2 -9305.922} C_VEL
LIN {X 0,Y 431.193,Z 654.285,A -85,B 0,C 180,E1 -9307.09,E2 -9307.09} C_VEL
LIN {X 0,Y 431.125,Z 655.342,A -85,B 0,C 180,E1 -9308.512,E2 -9308.512} C_VEL
LIN {X 0,Y 431.112,Z 655.8,A -85,B 0,C 180,E1 -9309.986,E2 -9309.986} C_VEL
LIN {X 0,Y 431.145,Z 655.261,A -85,B 0,C 180,E1 -9311.939,E2 -9311.939} C_VEL
LIN {X 0,Y 431.242,Z 654.289,A -85,B 0,C 180,E1 -9313.195,E2 -9313.195} C_VEL
LIN {X 0,Y 431.345,Z 652.711,A -85,B 0,C 180,E1 -9314.476,E2 -9314.476} C_VEL
LIN {X 0,Y 431.577,Z 649.514,A -85,B 0,C 180,E1 -9316.321,E2 -9316.321} C_VEL
LIN {X 0,Y 431.914,Z 644.232,A -85,B 0,C 180,E1 -9318.461,E2 -9318.461} C_VEL
LIN {X 0,Y 432.352,Z 638.45,A -85,B 0,C 180,E1 -9320.258,E2 -9320.258} C_VEL
LIN {X 0,Y 432.89,Z 631.876,A -85,B 0,C 180,E1 -9321.907,E2 -9321.907} C_VEL
LIN {X 0,Y 433.702,Z 623.376,A -85,B 0,C 180,E1 -9323.658,E2 -9323.658} C_VEL
LIN {X 0,Y 434.535,Z 614.103,A -85,B 0,C 180,E1 -9325.241,E2 -9325.241} C_VEL
LIN {X 0,Y 435.555,Z 603.665,A -85,B 0,C 180,E1 -9326.727,E2 -9326.727} C_VEL
LIN {X 0,Y 436.602,Z 592.362,A -85,B 0,C 180,E1 -9328.074,E2 -9328.074} C_VEL
LIN {X 0,Y 437.693,Z 579.808,A -85,B 0,C 180,E1 -9329.318,E2 -9329.318} C_VEL
LIN {X 0,Y 438.786,Z 566.969,A -85,B 0,C 180,E1 -9330.361,E2 -9330.361} C_VEL
LIN {X 0,Y 439.702,Z 553.089,A -85,B 0,C 180,E1 -9331.281,E2 -9331.281} C_VEL
LIN {X 0,Y 440.461,Z 539.637,A -85,B 0,C 180,E1 -9331.984,E2 -9331.984} C_VEL
LIN {X 0,Y 441.077,Z 524.499,A -85,B 0,C 180,E1 -9332.582,E2 -9332.582} C_VEL
LIN {X 0,Y 441.583,Z 508.709,A -85,B 0,C 180,E1 -9332.998,E2 -9332.998} C_VEL
LIN {X 0,Y 444.099,Z 373.604,A -85,B 0,C 180,E1 -9335.356,E2 -9335.356} C_VEL
LIN {X 0,Y 435.968,Z 355.154,A -85,B 0,C 180,E1 -9336.265,E2 -9336.265} C_VEL
LIN {X 0,Y 432.988,Z 348.873,A -85,B 0,C 180,E1 -9336.63,E2 -9336.63} C_VEL
LIN {X 0,Y 432.337,Z 346.256,A -85,B 0,C 180,E1 -9337.282,E2 -9337.282} C_VEL
LIN {X 0,Y 432.389,Z 346.246,A -85,B 0,C 180,E1 -9340.515,E2 -9340.515} C_VEL
LIN {X 0,Y 432.392,Z 346.254,A -85,B 0,C 180,E1 -9343.959,E2 -9343.959} C_VEL
LIN {X 0,Y 432.462,Z 346.242,A -85,B 0,C 180,E1 -9347.803,E2 -9347.803} C_VEL
LIN {X 0,Y 432.465,Z 346.242,A -85,B 0,C 180,E1 -9351.589,E2 -9351.589} C_VEL
LIN {X 0,Y 432.556,Z 346.227,A -85,B 0,C 180,E1 -9354.405,E2 -9354.405} C_VEL
LIN {X 0,Y 432.599,Z 346.223,A -85,B 0,C 180,E1 -9358.138,E2 -9358.138} C_VEL
LIN {X 0,Y 432.728,Z 346.208,A -85,B 0,C 180,E1 -9360,E2 -9360} C_VEL
LIN {X 0,Y 432.586,Z 346.223,A -85,B 0,C 180,E1 -9362.793,E2 -9362.793} C_VEL
LIN {X 0,Y 432.581,Z 346.229,A -85,B 0,C 180,E1 -9365.594,E2 -9365.594} C_VEL
LIN {X 0,Y 432.466,Z 346.238,A -85,B 0,C 180,E1 -9368.41,E2 -9368.41} C_VEL
LIN {X 0,Y 432.462,Z 346.237,A -85,B 0,C 180,E1 -9372.196,E2 -9372.196} C_VEL
LIN {X 0,Y 432.432,Z 346.24,A -85,B 0,C 180,E1 -9376.038,E2 -9376.038} C_VEL
LIN {X 0,Y 432.389,Z 346.251,A -85,B 0,C 180,E1 -9379.485,E2 -9379.485} C_VEL
LIN {X 0,Y 432.321,Z 346.259,A -85,B 0,C 180,E1 -9382.964,E2 -9382.964} C_VEL
LIN {X 0,Y 432.366,Z 346.25,A -85,B 0,C 180,E1 -9386.032,E2 -9386.032} C_VEL
LIN {X 0,Y 432.345,Z 346.255,A -85,B 0,C 180,E1 -9389.187,E2 -9389.187} C_VEL
LIN {X 0,Y 432.325,Z 346.255,A -85,B 0,C 180,E1 -9392.443,E2 -9392.443} C_VEL
LIN {X 0,Y 432.345,Z 346.256,A -85,B 0,C 180,E1 -9395.631,E2 -9395.631} C_VEL
LIN {X 0,Y 432.352,Z 346.256,A -85,B 0,C 180,E1 -9399.342,E2 -9399.342} C_VEL
LIN {X 0,Y 432.335,Z 346.256,A -85,B 0,C 180,E1 -9401.797,E2 -9401.797} C_VEL
LIN {X 0,Y 432.335,Z 346.257,A -85,B 0,C 180,E1 -9404.347,E2 -9404.347} C_VEL
LIN {X 0,Y 432.326,Z 346.261,A -85,B 0,C 180,E1 -9407.015,E2 -9407.015} C_VEL
LIN {X 0,Y 432.343,Z 346.257,A -85,B 0,C 180,E1 -9409.819,E2 -9409.819} C_VEL
LIN {X 0,Y 432.312,Z 346.258,A -85,B 0,C 180,E1 -9413.022,E2 -9413.022} C_VEL
LIN {X 0,Y 432.359,Z 346.271,A -85,B 0,C 180,E1 -9416.28,E2 -9416.28} C_VEL
LIN {X 0,Y 436.613,Z 362.297,A -85,B 0,C 180,E1 -9419.265,E2 -9419.265} C_VEL
LIN {X 0,Y 438.687,Z 372.391,A -85,B 0,C 180,E1 -9421.012,E2 -9421.012} C_VEL
LIN {X 0,Y 437.375,Z 390.38,A -85,B 0,C 180,E1 -9423.722,E2 -9423.722} C_VEL
LIN {X 0,Y 443.196,Z 422.27,A -85,B 0,C 180,E1 -9424.709,E2 -9424.709} C_VEL
LIN {X 0,Y 443.403,Z 427.508,A -85,B 0,C 180,E1 -9424.82,E2 -9424.82} C_VEL
LIN {X 0,Y 441.015,Z 558.668,A -85,B 0,C 180,E1 -9427.111,E2 -9427.111} C_VEL
LIN {X 0,Y 440.249,Z 574.769,A -85,B 0,C 180,E1 -9427.58,E2 -9427.58} C_VEL
LIN {X 0,Y 439.353,Z 589.802,A -85,B 0,C 180,E1 -9428.21,E2 -9428.21} C_VEL
LIN {X 0,Y 438.386,Z 603.78,A -85,B 0,C 180,E1 -9428.979,E2 -9428.979} C_VEL
LIN {X 0,Y 437.276,Z 617.242,A -85,B 0,C 180,E1 -9429.907,E2 -9429.907} C_VEL
LIN {X 0,Y 436.059,Z 630.977,A -85,B 0,C 180,E1 -9431.073,E2 -9431.073} C_VEL
LIN {X 0,Y 434.925,Z 644.088,A -85,B 0,C 180,E1 -9432.437,E2 -9432.437} C_VEL
LIN {X 0,Y 434.033,Z 654.889,A -85,B 0,C 180,E1 -9433.78,E2 -9433.78} C_VEL
LIN {X 0,Y 433.038,Z 665.992,A -85,B 0,C 180,E1 -9435.43,E2 -9435.43} C_VEL
LIN {X 0,Y 432.385,Z 675.137,A -85,B 0,C 180,E1 -9437.065,E2 -9437.065} C_VEL
LIN {X 0,Y 431.949,Z 682.926,A -85,B 0,C 180,E1 -9438.741,E2 -9438.741} C_VEL
LIN {X 0,Y 431.52,Z 690.116,A -85,B 0,C 180,E1 -9440.626,E2 -9440.626} C_VEL
LIN {X 0,Y 431.38,Z 695.786,A -85,B 0,C 180,E1 -9442.511,E2 -9442.511} C_VEL
LIN {X 0,Y 431.259,Z 700.077,A -85,B 0,C 180,E1 -9444.388,E2 -9444.388} C_VEL
LIN {X 0,Y 431.223,Z 703.094,A -85,B 0,C 180,E1 -9446.262,E2 -9446.262} C_VEL
LIN {X 0,Y 431.285,Z 704.907,A -85,B 0,C 180,E1 -9448.132,E2 -9448.132} C_VEL
LIN {X 0,Y 431.275,Z 705.543,A -85,B 0,C 180,E1 -9450,E2 -9450} C_VEL
LIN {X 0,Y 431.283,Z 704.953,A -85,B 0,C 180,E1 -9451.867,E2 -9451.867} C_VEL
LIN {X 0,Y 431.222,Z 703.174,A -85,B 0,C 180,E1 -9453.737,E2 -9453.737} C_VEL
LIN {X 0,Y 431.251,Z 700.192,A -85,B 0,C 180,E1 -9455.611,E2 -9455.611} C_VEL
LIN {X 0,Y 431.336,Z 695.934,A -85,B 0,C 180,E1 -9457.489,E2 -9457.489} C_VEL
LIN {X 0,Y 431.52,Z 690.289,A -85,B 0,C 180,E1 -9459.373,E2 -9459.373} C_VEL
LIN {X 0,Y 431.957,Z 683.113,A -85,B 0,C 180,E1 -9461.258,E2 -9461.258} C_VEL
LIN {X 0,Y 432.355,Z 675.799,A -85,B 0,C 180,E1 -9462.843,E2 -9462.843} C_VEL
LIN {X 0,Y 433.084,Z 666.184,A -85,B 0,C 180,E1 -9464.568,E2 -9464.568} C_VEL
LIN {X 0,Y 434.065,Z 655.016,A -85,B 0,C 180,E1 -9466.218,E2 -9466.218} C_VEL
LIN {X 0,Y 434.964,Z 644.028,A -85,B 0,C 180,E1 -9467.58,E2 -9467.58} C_VEL
LIN {X 0,Y 435.948,Z 632.19,A -85,B 0,C 180,E1 -9468.809,E2 -9468.809} C_VEL
LIN {X 0,Y 437.131,Z 618.544,A -85,B 0,C 180,E1 -9469.977,E2 -9469.977} C_VEL
LIN {X 0,Y 438.172,Z 605.136,A -85,B 0,C 180,E1 -9470.908,E2 -9470.908} C_VEL
LIN {X 0,Y 439.323,Z 589.816,A -85,B 0,C 180,E1 -9471.746,E2 -9471.746} C_VEL
LIN {X 0,Y 440.097,Z 574.419,A -85,B 0,C 180,E1 -9472.379,E2 -9472.379} C_VEL
LIN {X 0,Y 440.737,Z 559.149,A -85,B 0,C 180,E1 -9472.81,E2 -9472.81} C_VEL
LIN {X 0,Y 442.929,Z 432.865,A -85,B 0,C 180,E1 -9474.98,E2 -9474.98} C_VEL
LIN {X 0,Y 442.911,Z 422.985,A -85,B 0,C 180,E1 -9475.161,E2 -9475.161} C_VEL
LIN {X 0,Y 437.313,Z 392.176,A -85,B 0,C 180,E1 -9476.063,E2 -9476.063} C_VEL
LIN {X 0,Y 438.69,Z 374.203,A -85,B 0,C 180,E1 -9478.725,E2 -9478.725} C_VEL
LIN {X 0,Y 438.449,Z 370.78,A -85,B 0,C 180,E1 -9479.267,E2 -9479.267} C_VEL
LIN {X 0,Y 435.135,Z 356.918,A -85,B 0,C 180,E1 -9481.662,E2 -9481.662} C_VEL
LIN {X 0,Y 432.365,Z 346.252,A -85,B 0,C 180,E1 -9483.606,E2 -9483.606} C_VEL
LIN {X 0,Y 432.304,Z 346.263,A -85,B 0,C 180,E1 -9486.978,E2 -9486.978} C_VEL
LIN {X 0,Y 432.334,Z 346.252,A -85,B 0,C 180,E1 -9490.18,E2 -9490.18} C_VEL
LIN {X 0,Y 432.32,Z 346.259,A -85,B 0,C 180,E1 -9493.06,E2 -9493.06} C_VEL
LIN {X 0,Y 432.338,Z 346.254,A -85,B 0,C 180,E1 -9495.663,E2 -9495.663} C_VEL
LIN {X 0,Y 432.331,Z 346.253,A -85,B 0,C 180,E1 -9498.398,E2 -9498.398} C_VEL
LIN {X 0,Y 432.342,Z 346.252,A -85,B 0,C 180,E1 -9501.851,E2 -9501.851} C_VEL
LIN {X 0,Y 432.338,Z 346.257,A -85,B 0,C 180,E1 -9505.323,E2 -9505.323} C_VEL
LIN {X 0,Y 432.318,Z 346.256,A -85,B 0,C 180,E1 -9508.654,E2 -9508.654} C_VEL
LIN {X 0,Y 432.378,Z 346.247,A -85,B 0,C 180,E1 -9511.877,E2 -9511.877} C_VEL
LIN {X 0,Y 432.348,Z 346.257,A -85,B 0,C 180,E1 -9514.999,E2 -9514.999} C_VEL
LIN {X 0,Y 432.354,Z 346.25,A -85,B 0,C 180,E1 -9518.046,E2 -9518.046} C_VEL
LIN {X 0,Y 432.383,Z 346.254,A -85,B 0,C 180,E1 -9521.03,E2 -9521.03} C_VEL
LIN {X 0,Y 432.428,Z 346.24,A -85,B 0,C 180,E1 -9523.961,E2 -9523.961} C_VEL
LIN {X 0,Y 432.456,Z 346.237,A -85,B 0,C 180,E1 -9527.804,E2 -9527.804} C_VEL
LIN {X 0,Y 432.489,Z 346.234,A -85,B 0,C 180,E1 -9531.591,E2 -9531.591} C_VEL
LIN {X 0,Y 432.591,Z 346.222,A -85,B 0,C 180,E1 -9534.406,E2 -9534.406} C_VEL
LIN {X 0,Y 432.603,Z 346.219,A -85,B 0,C 180,E1 -9538.138,E2 -9538.138} C_VEL
LIN {X 0,Y 432.731,Z 346.203,A -85,B 0,C 180,E1 -9540,E2 -9540} C_VEL
LIN {X 0,Y 432.602,Z 346.225,A -85,B 0,C 180,E1 -9542.794,E2 -9542.794} C_VEL
LIN {X 0,Y 432.572,Z 346.226,A -85,B 0,C 180,E1 -9546.531,E2 -9546.531} C_VEL
LIN {X 0,Y 432.441,Z 346.241,A -85,B 0,C 180,E1 -9549.354,E2 -9549.354} C_VEL
LIN {X 0,Y 432.429,Z 346.248,A -85,B 0,C 180,E1 -9552.804,E2 -9552.804} C_VEL
LIN {X 0,Y 432.411,Z 346.246,A -85,B 0,C 180,E1 -9556.479,E2 -9556.479} C_VEL
LIN {X 0,Y 432.337,Z 346.252,A -85,B 0,C 180,E1 -9559.961,E2 -9559.961} C_VEL
LIN {X 0,Y 432.317,Z 346.259,A -85,B 0,C 180,E1 -9562.965,E2 -9562.965} C_VEL
LIN {X 0,Y 432.342,Z 346.255,A -85,B 0,C 180,E1 -9565.002,E2 -9565.002} C_VEL
LIN {X 0,Y 432.379,Z 346.248,A -85,B 0,C 180,E1 -9568.124,E2 -9568.124} C_VEL
LIN {X 0,Y 432.32,Z 346.255,A -85,B 0,C 180,E1 -9571.347,E2 -9571.347} C_VEL
LIN {X 0,Y 432.34,Z 346.259,A -85,B 0,C 180,E1 -9574.678,E2 -9574.678} C_VEL
LIN {X 0,Y 432.333,Z 346.254,A -85,B 0,C 180,E1 -9578.151,E2 -9578.151} C_VEL
LIN {X 0,Y 432.324,Z 346.253,A -85,B 0,C 180,E1 -9581.601,E2 -9581.601} C_VEL
LIN {X 0,Y 432.333,Z 346.257,A -85,B 0,C 180,E1 -9584.348,E2 -9584.348} C_VEL
LIN {X 0,Y 432.316,Z 346.257,A -85,B 0,C 180,E1 -9587.017,E2 -9587.017} C_VEL
LIN {X 0,Y 432.332,Z 346.253,A -85,B 0,C 180,E1 -9589.822,E2 -9589.822} C_VEL
LIN {X 0,Y 432.305,Z 346.258,A -85,B 0,C 180,E1 -9593.022,E2 -9593.022} C_VEL
LIN {X 0,Y 432.36,Z 346.251,A -85,B 0,C 180,E1 -9595.997,E2 -9595.997} C_VEL
LIN {X 0,Y 432.348,Z 346.25,A -85,B 0,C 180,E1 -9599.491,E2 -9599.491} C_VEL
LIN {X 0,Y 432.345,Z 346.252,A -85,B 0,C 180,E1 -9601.875,E2 -9601.875} C_VEL
LIN {X 0,Y 432.379,Z 346.247,A -85,B 0,C 180,E1 -9605.539,E2 -9605.539} C_VEL
LIN {X 0,Y 432.352,Z 346.251,A -85,B 0,C 180,E1 -9609.047,E2 -9609.047} C_VEL
LIN {X 0,Y 432.352,Z 346.253,A -85,B 0,C 180,E1 -9612.011,E2 -9612.011} C_VEL
LIN {X 0,Y 432.353,Z 346.251,A -85,B 0,C 180,E1 -9614.925,E2 -9614.925} C_VEL
LIN {X 0,Y 432.463,Z 346.238,A -85,B 0,C 180,E1 -9617.804,E2 -9617.804} C_VEL
LIN {X 0,Y 432.466,Z 346.236,A -85,B 0,C 180,E1 -9621.59,E2 -9621.59} C_VEL
LIN {X 0,Y 432.574,Z 346.229,A -85,B 0,C 180,E1 -9624.406,E2 -9624.406} C_VEL
LIN {X 0,Y 432.6,Z 346.225,A -85,B 0,C 180,E1 -9628.138,E2 -9628.138} C_VEL
LIN {X 0,Y 432.519,Z 346.23,A -85,B 0,C 180,E1 -9630.991,E2 -9630.991} C_VEL
LIN {X 0,Y 432.56,Z 346.226,A -85,B 0,C 180,E1 -9632.794,E2 -9632.794} C_VEL
LIN {X 0,Y 432.433,Z 346.24,A -85,B 0,C 180,E1 -9635.028,E2 -9635.028} C_VEL
LIN {X 0,Y 431.861,Z 346.315,A -85,B 0,C 180,E1 -9635.807,E2 -9635.807} C_VEL
LIN {X 0,Y 429.005,Z 346.67,A -85,B 0,C 180,E1 -9637.071,E2 -9637.071} C_VEL
LIN {X 0,Y 426.527,Z 346.982,A -85,B 0,C 180,E1 -9638.091,E2 -9638.091} C_VEL
LIN {X 0,Y 425.46,Z 347.109,A -85,B 0,C 180,E1 -9638.881,E2 -9638.881} C_VEL
LIN {X 0,Y 425.376,Z 347.119,A -85,B 0,C 180,E1 -9639.149,E2 -9639.149} C_VEL
LIN {X 0,Y 425.389,Z 347.119,A -85,B 0,C 180,E1 -9642.898,E2 -9642.898} C_VEL
LIN {X 0,Y 425.384,Z 347.318,A -85,B 0,C 180,E1 -9643.271,E2 -9643.271} C_VEL
LIN {X 0,Y 426.458,Z 350.168,A -85,B 0,C 180,E1 -9643.4,E2 -9643.4} C_VEL
LIN {X 0,Y 434.467,Z 368.558,A -85,B 0,C 180,E1 -9644.259,E2 -9644.259} C_VEL
LIN {X 0,Y 437.011,Z 374.721,A -85,B 0,C 180,E1 -9644.531,E2 -9644.531} C_VEL
LIN {X 0,Y 434.558,Z 512.124,A -85,B 0,C 180,E1 -9646.943,E2 -9646.943} C_VEL
LIN {X 0,Y 434.032,Z 527.079,A -85,B 0,C 180,E1 -9647.384,E2 -9647.384} C_VEL
LIN {X 0,Y 433.324,Z 541.904,A -85,B 0,C 180,E1 -9648.01,E2 -9648.01} C_VEL
LIN {X 0,Y 432.408,Z 556.825,A -85,B 0,C 180,E1 -9648.847,E2 -9648.847} C_VEL
LIN {X 0,Y 431.436,Z 570.047,A -85,B 0,C 180,E1 -9649.783,E2 -9649.783} C_VEL
LIN {X 0,Y 430.273,Z 583.333,A -85,B 0,C 180,E1 -9650.935,E2 -9650.935} C_VEL
LIN {X 0,Y 429.201,Z 595.758,A -85,B 0,C 180,E1 -9652.251,E2 -9652.251} C_VEL
LIN {X 0,Y 428.101,Z 606.891,A -85,B 0,C 180,E1 -9653.665,E2 -9653.665} C_VEL
LIN {X 0,Y 427.147,Z 616.886,A -85,B 0,C 180,E1 -9655.184,E2 -9655.184} C_VEL
LIN {X 0,Y 426.386,Z 625.504,A -85,B 0,C 180,E1 -9656.748,E2 -9656.748} C_VEL
LIN {X 0,Y 425.6,Z 634.046,A -85,B 0,C 180,E1 -9658.613,E2 -9658.613} C_VEL
LIN {X 0,Y 425.122,Z 640.031,A -85,B 0,C 180,E1 -9660.209,E2 -9660.209} C_VEL
LIN {X 0,Y 424.739,Z 645.433,A -85,B 0,C 180,E1 -9661.972,E2 -9661.972} C_VEL
LIN {X 0,Y 424.39,Z 650.381,A -85,B 0,C 180,E1 -9664.104,E2 -9664.104} C_VEL
LIN {X 0,Y 424.201,Z 653.116,A -85,B 0,C 180,E1 -9665.726,E2 -9665.726} C_VEL
LIN {X 0,Y 424.076,Z 655.351,A -85,B 0,C 180,E1 -9667.82,E2 -9667.82} C_VEL
LIN {X 0,Y 424.027,Z 656.024,A -85,B 0,C 180,E1 -9669.038,E2 -9669.038} C_VEL
LIN {X 0,Y 424.043,Z 656.188,A -85,B 0,C 180,E1 -9670.324,E2 -9670.324} C_VEL
LIN {X 0,Y 424.052,Z 655.773,A -85,B 0,C 180,E1 -9671.771,E2 -9671.771} C_VEL
LIN {X 0,Y 424.157,Z 654.765,A -85,B 0,C 180,E1 -9673.193,E2 -9673.193} C_VEL
LIN {X 0,Y 424.384,Z 651.845,A -85,B 0,C 180,E1 -9675.406,E2 -9675.406} C_VEL
LIN {X 0,Y 424.672,Z 648.106,A -85,B 0,C 180,E1 -9677.271,E2 -9677.271} C_VEL
LIN {X 0,Y 424.975,Z 643.279,A -85,B 0,C 180,E1 -9679.083,E2 -9679.083} C_VEL
LIN {X 0,Y 425.556,Z 636.308,A -85,B 0,C 180,E1 -9681.129,E2 -9681.129} C_VEL
LIN {X 0,Y 426.342,Z 628.224,A -85,B 0,C 180,E1 -9683.009,E2 -9683.009} C_VEL
LIN {X 0,Y 427.123,Z 619.969,A -85,B 0,C 180,E1 -9684.589,E2 -9684.589} C_VEL
LIN {X 0,Y 428.086,Z 610.774,A -85,B 0,C 180,E1 -9686.069,E2 -9686.069} C_VEL
LIN {X 0,Y 429.226,Z 599.835,A -85,B 0,C 180,E1 -9687.547,E2 -9687.547} C_VEL
LIN {X 0,Y 430.334,Z 587.823,A -85,B 0,C 180,E1 -9688.903,E2 -9688.903} C_VEL
LIN {X 0,Y 431.501,Z 574.573,A -85,B 0,C 180,E1 -9690.134,E2 -9690.134} C_VEL
LIN {X 0,Y 432.685,Z 560.477,A -85,B 0,C 180,E1 -9691.189,E2 -9691.189} C_VEL
LIN {X 0,Y 433.47,Z 547.87,A -85,B 0,C 180,E1 -9691.953,E2 -9691.953} C_VEL
LIN {X 0,Y 434.279,Z 532.864,A -85,B 0,C 180,E1 -9692.657,E2 -9692.657} C_VEL
LIN {X 0,Y 434.854,Z 517.477,A -85,B 0,C 180,E1 -9693.175,E2 -9693.175} C_VEL
LIN {X 0,Y 435.332,Z 497.866,A -85,B 0,C 180,E1 -9693.578,E2 -9693.578} C_VEL
LIN {X 0,Y 437.713,Z 375.338,A -85,B 0,C 180,E1 -9695.75,E2 -9695.75} C_VEL
LIN {X 0,Y 429.537,Z 357.063,A -85,B 0,C 180,E1 -9696.687,E2 -9696.687} C_VEL
LIN {X 0,Y 425.817,Z 349.428,A -85,B 0,C 180,E1 -9697.145,E2 -9697.145} C_VEL
LIN {X 0,Y 425.295,Z 347.136,A -85,B 0,C 180,E1 -9697.73,E2 -9697.73} C_VEL
LIN {X 0,Y 425.363,Z 347.121,A -85,B 0,C 180,E1 -9700.704,E2 -9700.704} C_VEL
LIN {X 0,Y 425.326,Z 347.13,A -85,B 0,C 180,E1 -9703.685,E2 -9703.685} C_VEL
LIN {X 0,Y 425.397,Z 347.122,A -85,B 0,C 180,E1 -9707.096,E2 -9707.096} C_VEL
LIN {X 0,Y 425.397,Z 347.119,A -85,B 0,C 180,E1 -9710.49,E2 -9710.49} C_VEL
LIN {X 0,Y 425.479,Z 347.11,A -85,B 0,C 180,E1 -9713.36,E2 -9713.36} C_VEL
LIN {X 0,Y 425.349,Z 347.126,A -85,B 0,C 180,E1 -9715.261,E2 -9715.261} C_VEL
LIN {X 0,Y 425.568,Z 347.099,A -85,B 0,C 180,E1 -9718.107,E2 -9718.107} C_VEL
LIN {X 0,Y 425.698,Z 347.084,A -85,B 0,C 180,E1 -9720,E2 -9720} C_VEL
LIN {X 0,Y 425.539,Z 347.101,A -85,B 0,C 180,E1 -9722.84,E2 -9722.84} C_VEL
LIN {X 0,Y 425.535,Z 347.106,A -85,B 0,C 180,E1 -9725.687,E2 -9725.687} C_VEL
LIN {X 0,Y 425.41,Z 347.117,A -85,B 0,C 180,E1 -9728.55,E2 -9728.55} C_VEL
LIN {X 0,Y 425.415,Z 347.114,A -85,B 0,C 180,E1 -9732.401,E2 -9732.401} C_VEL
LIN {X 0,Y 425.39,Z 347.116,A -85,B 0,C 180,E1 -9736.311,E2 -9736.311} C_VEL
LIN {X 0,Y 425.33,Z 347.129,A -85,B 0,C 180,E1 -9739.635,E2 -9739.635} C_VEL
LIN {X 0,Y 425.309,Z 347.132,A -85,B 0,C 180,E1 -9743.365,E2 -9743.365} C_VEL
LIN {X 0,Y 425.349,Z 347.126,A -85,B 0,C 180,E1 -9746.844,E2 -9746.844} C_VEL
LIN {X 0,Y 425.293,Z 347.13,A -85,B 0,C 180,E1 -9749.719,E2 -9749.719} C_VEL
LIN {X 0,Y 425.284,Z 347.136,A -85,B 0,C 180,E1 -9753.048,E2 -9753.048} C_VEL
LIN {X 0,Y 425.284,Z 347.135,A -85,B 0,C 180,E1 -9755.928,E2 -9755.928} C_VEL
LIN {X 0,Y 425.299,Z 347.134,A -85,B 0,C 180,E1 -9759.043,E2 -9759.043} C_VEL
LIN {X 0,Y 425.276,Z 347.138,A -85,B 0,C 180,E1 -9762.653,E2 -9762.653} C_VEL
LIN {X 0,Y 425.269,Z 347.136,A -85,B 0,C 180,E1 -9766.045,E2 -9766.045} C_VEL
LIN {X 0,Y 425.286,Z 347.138,A -85,B 0,C 180,E1 -9769.479,E2 -9769.479} C_VEL
LIN {X 0,Y 425.281,Z 347.138,A -85,B 0,C 180,E1 -9772.488,E2 -9772.488} C_VEL
LIN {X 0,Y 425.337,Z 347.235,A -85,B 0,C 180,E1 -9775.837,E2 -9775.837} C_VEL
LIN {X 0,Y 429.311,Z 362.1,A -85,B 0,C 180,E1 -9778.685,E2 -9778.685} C_VEL
LIN {X 0,Y 431.889,Z 373.789,A -85,B 0,C 180,E1 -9780.778,E2 -9780.778} C_VEL
LIN {X 0,Y 431.095,Z 385.436,A -85,B 0,C 180,E1 -9782.577,E2 -9782.577} C_VEL
LIN {X 0,Y 430.751,Z 390.237,A -85,B 0,C 180,E1 -9783.267,E2 -9783.267} C_VEL
LIN {X 0,Y 436.073,Z 419.1,A -85,B 0,C 180,E1 -9784.193,E2 -9784.193} C_VEL
LIN {X 0,Y 437.07,Z 425.478,A -85,B 0,C 180,E1 -9784.381,E2 -9784.381} C_VEL
LIN {X 0,Y 434.506,Z 557.495,A -85,B 0,C 180,E1 -9786.717,E2 -9786.717} C_VEL
LIN {X 0,Y 433.776,Z 573.395,A -85,B 0,C 180,E1 -9787.177,E2 -9787.177} C_VEL
LIN {X 0,Y 432.844,Z 588.213,A -85,B 0,C 180,E1 -9787.793,E2 -9787.793} C_VEL
LIN {X 0,Y 431.737,Z 603.449,A -85,B 0,C 180,E1 -9788.639,E2 -9788.639} C_VEL
LIN {X 0,Y 430.573,Z 616.874,A -85,B 0,C 180,E1 -9789.58,E2 -9789.58} C_VEL
LIN {X 0,Y 429.297,Z 630.581,A -85,B 0,C 180,E1 -9790.763,E2 -9790.763} C_VEL
LIN {X 0,Y 428.113,Z 643.651,A -85,B 0,C 180,E1 -9792.143,E2 -9792.143} C_VEL
LIN {X 0,Y 427.138,Z 654.489,A -85,B 0,C 180,E1 -9793.511,E2 -9793.511} C_VEL
LIN {X 0,Y 426.094,Z 665.59,A -85,B 0,C 180,E1 -9795.187,E2 -9795.187} C_VEL
LIN {X 0,Y 425.371,Z 675.023,A -85,B 0,C 180,E1 -9796.906,E2 -9796.906} C_VEL
LIN {X 0,Y 424.873,Z 682.52,A -85,B 0,C 180,E1 -9798.551,E2 -9798.551} C_VEL
LIN {X 0,Y 424.435,Z 689.704,A -85,B 0,C 180,E1 -9800.468,E2 -9800.468} C_VEL
LIN {X 0,Y 424.302,Z 695.373,A -85,B 0,C 180,E1 -9802.385,E2 -9802.385} C_VEL
LIN {X 0,Y 424.174,Z 699.667,A -85,B 0,C 180,E1 -9804.294,E2 -9804.294} C_VEL
LIN {X 0,Y 424.128,Z 702.685,A -85,B 0,C 180,E1 -9806.199,E2 -9806.199} C_VEL
LIN {X 0,Y 424.249,Z 703.745,A -85,B 0,C 180,E1 -9807.151,E2 -9807.151} C_VEL
LIN {X 0,Y 424.187,Z 704.961,A -85,B 0,C 180,E1 -9809.05,E2 -9809.05} C_VEL
LIN {X 0,Y 424.187,Z 704.99,A -85,B 0,C 180,E1 -9810.949,E2 -9810.949} C_VEL
LIN {X 0,Y 424.243,Z 703.802,A -85,B 0,C 180,E1 -9812.848,E2 -9812.848} C_VEL
LIN {X 0,Y 424.158,Z 701.417,A -85,B 0,C 180,E1 -9814.752,E2 -9814.752} C_VEL
LIN {X 0,Y 424.209,Z 697.799,A -85,B 0,C 180,E1 -9816.659,E2 -9816.659} C_VEL
LIN {X 0,Y 424.366,Z 692.854,A -85,B 0,C 180,E1 -9818.571,E2 -9818.571} C_VEL
LIN {X 0,Y 424.642,Z 686.449,A -85,B 0,C 180,E1 -9820.489,E2 -9820.489} C_VEL
LIN {X 0,Y 425.125,Z 678.41,A -85,B 0,C 180,E1 -9822.41,E2 -9822.41} C_VEL
LIN {X 0,Y 425.819,Z 669.848,A -85,B 0,C 180,E1 -9824.089,E2 -9824.089} C_VEL
LIN {X 0,Y 426.479,Z 661.145,A -85,B 0,C 180,E1 -9825.532,E2 -9825.532} C_VEL
LIN {X 0,Y 427.501,Z 650.858,A -85,B 0,C 180,E1 -9826.966,E2 -9826.966} C_VEL
LIN {X 0,Y 428.497,Z 638.616,A -85,B 0,C 180,E1 -9828.404,E2 -9828.404} C_VEL
LIN {X 0,Y 429.589,Z 626.363,A -85,B 0,C 180,E1 -9829.595,E2 -9829.595} C_VEL
LIN {X 0,Y 430.765,Z 613.07,A -85,B 0,C 180,E1 -9830.659,E2 -9830.659} C_VEL
LIN {X 0,Y 431.821,Z 600.457,A -85,B 0,C 180,E1 -9831.481,E2 -9831.481} C_VEL
LIN {X 0,Y 432.788,Z 585.872,A -85,B 0,C 180,E1 -9832.239,E2 -9832.239} C_VEL
LIN {X 0,Y 433.646,Z 570.407,A -85,B 0,C 180,E1 -9832.832,E2 -9832.832} C_VEL
LIN {X 0,Y 434.236,Z 554.708,A -85,B 0,C 180,E1 -9833.235,E2 -9833.235} C_VEL
LIN {X 0,Y 436.399,Z 434.245,A -85,B 0,C 180,E1 -9835.328,E2 -9835.328} C_VEL
LIN {X 0,Y 436.413,Z 424.091,A -85,B 0,C 180,E1 -9835.516,E2 -9835.516} C_VEL
LIN {X 0,Y 430.586,Z 391.806,A -85,B 0,C 180,E1 -9836.481,E2 -9836.481} C_VEL
LIN {X 0,Y 431.916,Z 375.216,A -85,B 0,C 180,E1 -9838.98,E2 -9838.98} C_VEL
LIN {X 0,Y 430.963,Z 369.684,A -85,B 0,C 180,E1 -9839.912,E2 -9839.912} C_VEL
LIN {X 0,Y 428.151,Z 358.057,A -85,B 0,C 180,E1 -9841.963,E2 -9841.963} C_VEL
LIN {X 0,Y 425.325,Z 347.129,A -85,B 0,C 180,E1 -9844.002,E2 -9844.002} C_VEL
LIN {X 0,Y 425.275,Z 347.139,A -85,B 0,C 180,E1 -9847.511,E2 -9847.511} C_VEL
LIN {X 0,Y 425.279,Z 347.132,A -85,B 0,C 180,E1 -9850.52,E2 -9850.52} C_VEL
LIN {X 0,Y 425.261,Z 347.139,A -85,B 0,C 180,E1 -9853.352,E2 -9853.352} C_VEL
LIN {X 0,Y 425.261,Z 347.135,A -85,B 0,C 180,E1 -9856.648,E2 -9856.648} C_VEL
LIN {X 0,Y 425.283,Z 347.131,A -85,B 0,C 180,E1 -9859.873,E2 -9859.873} C_VEL
LIN {X 0,Y 425.281,Z 347.132,A -85,B 0,C 180,E1 -9862.487,E2 -9862.487} C_VEL
LIN {X 0,Y 425.305,Z 347.129,A -85,B 0,C 180,E1 -9865.817,E2 -9865.817} C_VEL
LIN {X 0,Y 425.287,Z 347.136,A -85,B 0,C 180,E1 -9869.239,E2 -9869.239} C_VEL
LIN {X 0,Y 425.345,Z 347.124,A -85,B 0,C 180,E1 -9872.442,E2 -9872.442} C_VEL
LIN {X 0,Y 425.348,Z 347.124,A -85,B 0,C 180,E1 -9875.602,E2 -9875.602} C_VEL
LIN {X 0,Y 425.29,Z 347.133,A -85,B 0,C 180,E1 -9878.682,E2 -9878.682} C_VEL
LIN {X 0,Y 425.33,Z 347.126,A -85,B 0,C 180,E1 -9881.703,E2 -9881.703} C_VEL
LIN {X 0,Y 425.346,Z 347.126,A -85,B 0,C 180,E1 -9884.671,E2 -9884.671} C_VEL
LIN {X 0,Y 425.409,Z 347.116,A -85,B 0,C 180,E1 -9887.598,E2 -9887.598} C_VEL
LIN {X 0,Y 425.44,Z 347.113,A -85,B 0,C 180,E1 -9891.45,E2 -9891.45} C_VEL
LIN {X 0,Y 425.547,Z 347.099,A -85,B 0,C 180,E1 -9894.313,E2 -9894.313} C_VEL
LIN {X 0,Y 425.573,Z 347.095,A -85,B 0,C 180,E1 -9898.108,E2 -9898.108} C_VEL
LIN {X 0,Y 425.701,Z 347.079,A -85,B 0,C 180,E1 -9900,E2 -9900} C_VEL
LIN {X 0,Y 425.553,Z 347.104,A -85,B 0,C 180,E1 -9902.84,E2 -9902.84} C_VEL
LIN {X 0,Y 425.53,Z 347.105,A -85,B 0,C 180,E1 -9906.639,E2 -9906.639} C_VEL
LIN {X 0,Y 425.399,Z 347.117,A -85,B 0,C 180,E1 -9909.51,E2 -9909.51} C_VEL
LIN {X 0,Y 425.391,Z 347.124,A -85,B 0,C 180,E1 -9912.904,E2 -9912.904} C_VEL
LIN {X 0,Y 425.36,Z 347.126,A -85,B 0,C 180,E1 -9916.605,E2 -9916.605} C_VEL
LIN {X 0,Y 425.327,Z 347.125,A -85,B 0,C 180,E1 -9919.636,E2 -9919.636} C_VEL
LIN {X 0,Y 425.286,Z 347.133,A -85,B 0,C 180,E1 -9922.339,E2 -9922.339} C_VEL
LIN {X 0,Y 425.32,Z 347.133,A -85,B 0,C 180,E1 -9924.658,E2 -9924.658} C_VEL
LIN {X 0,Y 425.344,Z 347.123,A -85,B 0,C 180,E1 -9927.558,E2 -9927.558} C_VEL
LIN {X 0,Y 425.287,Z 347.136,A -85,B 0,C 180,E1 -9930.817,E2 -9930.817} C_VEL
LIN {X 0,Y 425.311,Z 347.13,A -85,B 0,C 180,E1 -9934.289,E2 -9934.289} C_VEL
LIN {X 0,Y 425.277,Z 347.131,A -85,B 0,C 180,E1 -9937.695,E2 -9937.695} C_VEL
LIN {X 0,Y 425.276,Z 347.138,A -85,B 0,C 180,E1 -9940.52,E2 -9940.52} C_VEL
LIN {X 0,Y 425.26,Z 347.134,A -85,B 0,C 180,E1 -9943.957,E2 -9943.957} C_VEL
LIN {X 0,Y 425.27,Z 347.132,A -85,B 0,C 180,E1 -9947.347,E2 -9947.347} C_VEL
LIN {X 0,Y 425.284,Z 347.131,A -85,B 0,C 180,E1 -9949.873,E2 -9949.873} C_VEL
LIN {X 0,Y 425.277,Z 347.139,A -85,B 0,C 180,E1 -9952.49,E2 -9952.49} C_VEL
LIN {X 0,Y 425.308,Z 347.128,A -85,B 0,C 180,E1 -9955.818,E2 -9955.818} C_VEL
LIN {X 0,Y 425.292,Z 347.13,A -85,B 0,C 180,E1 -9959.24,E2 -9959.24} C_VEL
LIN {X 0,Y 425.272,Z 347.139,A -85,B 0,C 180,E1 -9962.437,E2 -9962.437} C_VEL
LIN {X 0,Y 425.348,Z 347.123,A -85,B 0,C 180,E1 -9965.602,E2 -9965.602} C_VEL
LIN {X 0,Y 425.296,Z 347.133,A -85,B 0,C 180,E1 -9968.682,E2 -9968.682} C_VEL
LIN {X 0,Y 425.317,Z 347.127,A -85,B 0,C 180,E1 -9971.702,E2 -9971.702} C_VEL
LIN {X 0,Y 425.307,Z 347.131,A -85,B 0,C 180,E1 -9974.67,E2 -9974.67} C_VEL
LIN {X 0,Y 425.416,Z 347.114,A -85,B 0,C 180,E1 -9977.599,E2 -9977.599} C_VEL
LIN {X 0,Y 425.41,Z 347.115,A -85,B 0,C 180,E1 -9981.45,E2 -9981.45} C_VEL
LIN {X 0,Y 425.529,Z 347.108,A -85,B 0,C 180,E1 -9984.313,E2 -9984.313} C_VEL
LIN {X 0,Y 425.569,Z 347.1,A -85,B 0,C 180,E1 -9988.108,E2 -9988.108} C_VEL
LIN {X 0,Y 425.483,Z 347.106,A -85,B 0,C 180,E1 -9990.947,E2 -9990.947} C_VEL
LIN {X 0,Y 425.515,Z 347.103,A -85,B 0,C 180,E1 -9992.841,E2 -9992.841} C_VEL
LIN {X 0,Y 425.513,Z 347.104,A -85,B 0,C 180,E1 -9995.688,E2 -9995.688} C_VEL
LIN {X 0,Y 425.399,Z 347.119,A -85,B 0,C 180,E1 -9998.551,E2 -9998.551} C_VEL
LIN {X 0,Y 425.376,Z 347.119,A -85,B 0,C 180,E1 -9999.149,E2 -9999.149} C_VEL
LIN {X 0,Y 424.699,Z 347.206,A -85,B 0,C 180,E1 -9999.676,E2 -9999.676} C_VEL
LIN {X 0,Y 421.843,Z 347.563,A -85,B 0,C 180,E1 -10000.499,E2 -10000.499} C_VEL
LIN {X 0,Y 418.976,Z 347.921,A -85,B 0,C 180,E1 -10001.334,E2 -10001.334} C_VEL
LIN {X 0,Y 418.304,Z 348.002,A -85,B 0,C 180,E1 -10001.873,E2 -10001.873} C_VEL
LIN {X 0,Y 418.351,Z 348.021,A -85,B 0,C 180,E1 -10002.82,E2 -10002.82} C_VEL
LIN {X 0,Y 419.473,Z 351.061,A -85,B 0,C 180,E1 -10002.956,E2 -10002.956} C_VEL
LIN {X 0,Y 427.453,Z 369.014,A -85,B 0,C 180,E1 -10003.827,E2 -10003.827} C_VEL
LIN {X 0,Y 430.567,Z 376.795,A -85,B 0,C 180,E1 -10004.173,E2 -10004.173} C_VEL
LIN {X 0,Y 427.995,Z 511.983,A -85,B 0,C 180,E1 -10006.578,E2 -10006.578} C_VEL
LIN {X 0,Y 427.456,Z 527.211,A -85,B 0,C 180,E1 -10007.03,E2 -10007.03} C_VEL
LIN {X 0,Y 426.692,Z 542.635,A -85,B 0,C 180,E1 -10007.692,E2 -10007.692} C_VEL
LIN {X 0,Y 425.75,Z 557.279,A -85,B 0,C 180,E1 -10008.528,E2 -10008.528} C_VEL
LIN {X 0,Y 424.673,Z 571.172,A -85,B 0,C 180,E1 -10009.533,E2 -10009.533} C_VEL
LIN {X 0,Y 423.511,Z 583.79,A -85,B 0,C 180,E1 -10010.649,E2 -10010.649} C_VEL
LIN {X 0,Y 422.382,Z 596.215,A -85,B 0,C 180,E1 -10011.986,E2 -10011.986} C_VEL
LIN {X 0,Y 421.24,Z 607.306,A -85,B 0,C 180,E1 -10013.418,E2 -10013.418} C_VEL
LIN {X 0,Y 420.185,Z 617.78,A -85,B 0,C 180,E1 -10015.039,E2 -10015.039} C_VEL
LIN {X 0,Y 419.269,Z 627.717,A -85,B 0,C 180,E1 -10016.91,E2 -10016.91} C_VEL
LIN {X 0,Y 418.497,Z 636.07,A -85,B 0,C 180,E1 -10018.85,E2 -10018.85} C_VEL
LIN {X 0,Y 417.98,Z 642.25,A -85,B 0,C 180,E1 -10020.612,E2 -10020.612} C_VEL
LIN {X 0,Y 417.531,Z 647.96,A -85,B 0,C 180,E1 -10022.688,E2 -10022.688} C_VEL
LIN {X 0,Y 417.266,Z 651.446,A -85,B 0,C 180,E1 -10024.38,E2 -10024.38} C_VEL
LIN {X 0,Y 417.074,Z 654.119,A -85,B 0,C 180,E1 -10026.142,E2 -10026.142} C_VEL
LIN {X 0,Y 416.989,Z 655.601,A -85,B 0,C 180,E1 -10027.613,E2 -10027.613} C_VEL
LIN {X 0,Y 416.945,Z 656.587,A -85,B 0,C 180,E1 -10029.832,E2 -10029.832} C_VEL
LIN {X 0,Y 416.956,Z 656.497,A -85,B 0,C 180,E1 -10031.1,E2 -10031.1} C_VEL
LIN {X 0,Y 417.012,Z 655.872,A -85,B 0,C 180,E1 -10032.387,E2 -10032.387} C_VEL
LIN {X 0,Y 417.112,Z 654.707,A -85,B 0,C 180,E1 -10033.695,E2 -10033.695} C_VEL
LIN {X 0,Y 417.343,Z 651.948,A -85,B 0,C 180,E1 -10035.684,E2 -10035.684} C_VEL
LIN {X 0,Y 417.655,Z 647.667,A -85,B 0,C 180,E1 -10037.766,E2 -10037.766} C_VEL
LIN {X 0,Y 418.075,Z 642.194,A -85,B 0,C 180,E1 -10039.745,E2 -10039.745} C_VEL
LIN {X 0,Y 418.714,Z 635.647,A -85,B 0,C 180,E1 -10041.608,E2 -10041.608} C_VEL
LIN {X 0,Y 419.441,Z 628.603,A -85,B 0,C 180,E1 -10043.245,E2 -10043.245} C_VEL
LIN {X 0,Y 420.377,Z 619.493,A -85,B 0,C 180,E1 -10045.005,E2 -10045.005} C_VEL
LIN {X 0,Y 421.441,Z 609.461,A -85,B 0,C 180,E1 -10046.611,E2 -10046.611} C_VEL
LIN {X 0,Y 422.606,Z 598.979,A -85,B 0,C 180,E1 -10048.01,E2 -10048.01} C_VEL
LIN {X 0,Y 423.734,Z 587.096,A -85,B 0,C 180,E1 -10049.346,E2 -10049.346} C_VEL
LIN {X 0,Y 424.862,Z 575.081,A -85,B 0,C 180,E1 -10050.467,E2 -10050.467} C_VEL
LIN {X 0,Y 426.079,Z 561.665,A -85,B 0,C 180,E1 -10051.49,E2 -10051.49} C_VEL
LIN {X 0,Y 426.925,Z 548.865,A -85,B 0,C 180,E1 -10052.286,E2 -10052.286} C_VEL
LIN {X 0,Y 427.761,Z 533.893,A -85,B 0,C 180,E1 -10053.007,E2 -10053.007} C_VEL
LIN {X 0,Y 428.345,Z 519.127,A -85,B 0,C 180,E1 -10053.524,E2 -10053.524} C_VEL
LIN {X 0,Y 428.845,Z 501.973,A -85,B 0,C 180,E1 -10053.9,E2 -10053.9} C_VEL
LIN {X 0,Y 431.366,Z 377.243,A -85,B 0,C 180,E1 -10056.155,E2 -10056.155} C_VEL
LIN {X 0,Y 424.098,Z 360.906,A -85,B 0,C 180,E1 -10057.016,E2 -10057.016} C_VEL
LIN {X 0,Y 418.743,Z 349.96,A -85,B 0,C 180,E1 -10057.682,E2 -10057.682} C_VEL
LIN {X 0,Y 418.258,Z 348.011,A -85,B 0,C 180,E1 -10058.183,E2 -10058.183} C_VEL
LIN {X 0,Y 418.273,Z 348.008,A -85,B 0,C 180,E1 -10061.382,E2 -10061.382} C_VEL
LIN {X 0,Y 418.256,Z 348.011,A -85,B 0,C 180,E1 -10064.404,E2 -10064.404} C_VEL
LIN {X 0,Y 418.359,Z 348,A -85,B 0,C 180,E1 -10067.385,E2 -10067.385} C_VEL
LIN {X 0,Y 418.338,Z 347.999,A -85,B 0,C 180,E1 -10070.328,E2 -10070.328} C_VEL
LIN {X 0,Y 418.444,Z 347.986,A -85,B 0,C 180,E1 -10073.248,E2 -10073.248} C_VEL
LIN {X 0,Y 418.32,Z 348.001,A -85,B 0,C 180,E1 -10075.181,E2 -10075.181} C_VEL
LIN {X 0,Y 418.537,Z 347.976,A -85,B 0,C 180,E1 -10078.075,E2 -10078.075} C_VEL
LIN {X 0,Y 418.667,Z 347.96,A -85,B 0,C 180,E1 -10080,E2 -10080} C_VEL
LIN {X 0,Y 418.495,Z 347.979,A -85,B 0,C 180,E1 -10082.887,E2 -10082.887} C_VEL
LIN {X 0,Y 418.492,Z 347.982,A -85,B 0,C 180,E1 -10085.783,E2 -10085.783} C_VEL
LIN {X 0,Y 418.38,Z 347.993,A -85,B 0,C 180,E1 -10088.695,E2 -10088.695} C_VEL
LIN {X 0,Y 418.317,Z 348.003,A -85,B 0,C 180,E1 -10091.631,E2 -10091.631} C_VEL
LIN {X 0,Y 418.304,Z 348.002,A -85,B 0,C 180,E1 -10094.597,E2 -10094.597} C_VEL
LIN {X 0,Y 418.282,Z 348.005,A -85,B 0,C 180,E1 -10097.604,E2 -10097.604} C_VEL
LIN {X 0,Y 418.252,Z 348.009,A -85,B 0,C 180,E1 -10100.663,E2 -10100.663} C_VEL
LIN {X 0,Y 418.29,Z 348.002,A -85,B 0,C 180,E1 -10103.781,E2 -10103.781} C_VEL
LIN {X 0,Y 418.312,Z 348.002,A -85,B 0,C 180,E1 -10107.07,E2 -10107.07} C_VEL
LIN {X 0,Y 418.246,Z 348.007,A -85,B 0,C 180,E1 -10110.272,E2 -10110.272} C_VEL
